END_VAR
VAR_INST
	boolEx				: BoolEx := (variable := _boolVariable);
	conditionTrueTimer	: Tc2_Standard.TON;
END_VAR
TcUnit.TEST('Test01_BooleanTrue_ExpectTrueAfterElapsedTime');

conditionTrueTimer();
IF NOT conditionTrueTimer.Q THEN
	_boolVariable := TRUE;
	conditionTrueTimer(IN := TRUE, PT := T#20MS);
	AssertFalse(
		Condition := boolEx.HasBeenTrueForAtLeast(T#20MS),
		Message := 'HasBeenTrueForAtLeast returned TRUE before elapsed time.');
ELSE
	AssertTrue(
		Condition := boolEx.HasBeenTrueForAtLeast(T#20MS),
		Message := 'HasBeenTrueForAtLeast returned FALSE after elapsed time.');
		TcUnit.TEST_FINISHED();
END_IF
END_METHOD

METHOD Test02_BooleanFalse_ExpectTrueAfterElapsedTime : BOOL
VAR_INST
	boolEx			: BoolEx := (variable := _boolVariable);
	conditionTimer	: Tc2_Standard.TON;
END_VAR
TcUnit.TEST('Test02_BooleanFalse_ExpectTrueAfterElapsedTime');
IF TcUnit.IS_TEST_FINISHED('Test01_BooleanTrue_ExpectTrueAfterElapsedTime') THEN
	_boolVariable := FALSE;
	conditionTimer();
	IF NOT conditionTimer.Q THEN
		conditionTimer(IN := TRUE, PT := T#20MS);
		AssertFalse(
			Condition := boolEx.HasBeenFalseForAtLeast(T#20MS),
			Message := 'HasBeenFalseForAtLeast returned TRUE before elapsed time.');
	ELSE
		AssertTrue(
			Condition := boolEx.HasBeenFalseForAtLeast(T#20MS),
			Message := 'HasBeenFalseForAtLeast returned FALSE after elapsed time.');
			TcUnit.TEST_FINISHED();
	END_IF
END_IF
END_METHOD

METHOD Test03_RisingAndFallingEdge_ExpectPulses
VAR_INPUT
END_VAR

VAR_INST
	boolEx : BoolEx := (variable := _boolVariable);
END_VAR
TcUnit.TEST('Test03_RisingAndFallingEdge_ExpectPulses');


IF TcUnit.IS_TEST_FINISHED('Test02_BooleanFalse_ExpectTrueAfterElapsedTime') THEN
	_boolVariable := FALSE;
	AssertFalse(
		Condition := boolEx.HasRisingEdge,
		Message := 'When value has not changed, the HasRisingEdge should be false');
	AssertFalse(
		Condition := boolEx.HasFallingEdge,
		Message := 'When value has not changed, the HasFallingEdge should be false');
	_boolVariable := TRUE;	
	AssertTrue(
		Condition := boolEx.HasRisingEdge,
		Message := 'When value has changed from FALSE to TRUE, the HasRisingEdge should be TRUE');
	AssertFalse(
		Condition := boolEx.HasFallingEdge,
		Message := 'When value has changed to TRUE, the HasFallingEdge should be false');
	_boolVariable := FALSE;
	AssertTrue(
		Condition := boolEx.HasFallingEdge,
		Message := 'When value has changed from TRUE to FALSE, the HasFallingEdge should be TRUE');
	AssertFalse(
		Condition := boolEx.HasRisingEdge,
		Message := 'When value has not changed, the HasRisingEdge should be false');
	AssertFalse(
		Condition := boolEx.HasFallingEdge,
		Message := 'When value has not changed, the HasRisingEdge should be false');	
	TcUnit.TEST_FINISHED();
	
END_IF
END_METHOD

METHOD Test04_GetAndSetValue
VAR_INPUT
END_VAR
VAR_INST
	boolEx	: BoolEx := (variable := _boolVariable);
END_VAR
TcUnit.TEST('Test04_GetAndSetValue');
IF TcUnit.IS_TEST_FINISHED('Test03_RisingAndFallingEdge_ExpectPulses') THEN
	_boolVariable := FALSE;
	boolEx.Value := TRUE;	
	AssertTrue(
		Condition := _boolVariable,
		Message := 'Setting value to TRUE failed');
		
	boolEx.Value := FALSE;
	AssertFalse(
		Condition := _boolVariable,
		Message := 'Setting value to FALSE failed');
		
	AssertEquals_BOOL(
		Actual := boolEx.Value,
		Expected := _boolVariable,
		Message := 'Value returned incorrect result.');
		
	_boolVariable := TRUE;
	AssertEquals_BOOL(
		Actual := boolEx.Value,
		Expected := _boolVariable,
		Message := 'Value returned incorrect result.');
	
	TcUnit.TEST_FINISHED();
END_IF
END_METHOD

METHOD Test05_Toggle_ExpectValueInverts
VAR_INPUT
END_VAR
TcUnit.TEST('Test05_Toggle_ExpectValueInverts');
IF TcUnit.IS_TEST_FINISHED('Test04_GetAndSetValue') THEN
	_boolEx.Value := FALSE;
	AssertFalse(
		Condition := _boolEx.Value,
		Message := 'Expected value to be false.');
		
	_boolEx.Toggle();
	AssertTrue(
		Condition := _boolEx.Value,
		Message := 'Toggle to TRUE failed');
		
	_boolEx.Toggle();
	AssertFalse(
		Condition := _boolEx.Value,
		Message := 'Toggle to FALSE failed');	
	TcUnit.TEST_FINISHED();
END_IF
END_METHOD

METHOD Test06_PulseWithInterval_100ms_ExpectValueChangeEvery100ms
VAR_INPUT
END_VAR
VAR_INST
	timerOn		: Tc2_Standard.TON;
	timerOff	: Tc2_Standard.TON;
END_VAR
TcUnit.TEST('Test06_PulseWithInterval_100ms_ExpectValueChangeEvery100ms');
IF TcUnit.IS_TEST_FINISHED('Test05_Toggle_ExpectValueInverts') THEN
	_boolEx.Value := FALSE;
	_boolEx.PulseWithInterval(durationOn := T#100MS, durationOff := T#50MS);
	timerOn(IN := TRUE, PT := T#100MS);
	IF NOT timerOn.Q THEN
		AssertTrue(
			Condition := _boolEx.Value,
			Message := 'Value should be TRUE until the durationOn expires.');
	ELSE
		timerOff(IN := TRUE, PT := T#50MS);
		IF timeroff.Q THEN
			AssertTrue(
				Condition := _boolEx.Value,
				Message := 'Value should be TRUE after the durationOff expires.');
			TcUnit.TEST_FINISHED();
			RETURN;
		END_IF
		AssertFalse(
			Condition := _boolEx.Value,
			Message := 'Value should be FALSE after durationOn expires.');

	END_IF
END_IF
END_METHOD

METHOD Test07_Set_ExpectTrue
VAR_INPUT
END_VAR
TcUnit.TEST('Test07_Set_ExpectTrue');

IF TcUnit.IS_TEST_FINISHED('Test06_PulseWithInterval_100ms_ExpectValueChangeEvery100ms') THEN 
	_boolEx.Value := FALSE;
	_boolEx.Set();
	AssertTrue(
		Condition := _boolEx.Value,
		Message := 'Set() did not set the value to TRUE.');
	TcUnit.TEST_FINISHED();
END_IF
END_METHOD

METHOD Test08_Reset_ExpectFalse
VAR_INPUT
END_VAR
TcUnit.TEST('Test08_Reset_ExpectFalse');

IF TcUnit.IS_TEST_FINISHED('Test07_Set_ExpectTrue') THEN 
	_boolEx.Value := TRUE;
	_boolEx.Reset();
	AssertFalse(
		Condition := _boolEx.Value,
		Message := 'Reset() did not set the value to FALSE.');
	TcUnit.TEST_FINISHED();
END_IF
END_METHOD

END_FUNCTION_BLOCK

// TESTS/Test suites/FB_DateTimeToStringConverter_Tests
FUNCTION_BLOCK INTERNAL FB_DateTimeToStringConverter_Tests EXTENDS FB_TestSuite
VAR_INPUT
END_VAR
VAR_OUTPUT
END_VAR
VAR
	_localSystemTime			: Tc2_Utilities.FB_LocalSystemTime;
	_dateTimeToStringConverter	: FB_DateTimeToStringConverter;
END_VAR

_localSystemTime(
	sNetID:= '', 
	bEnable:= TRUE, 
	dwCycle:= 1);
	
_dateTimeToStringConverter(localSystemTime := _localSystemTime);

Test01_Year();
Test02_Month();
Test03_Day();
Test04_Hour();
Test05_Minute();
Test06_Second();
Test07_Millisecond();

METHOD Test01_Year
VAR_INPUT
END_VAR
TcUnit.TEST('Test01_Year');

AssertEquals_STRING(
	Actual := _dateTimeToStringConverter.Year(),
	Expected := WORD_TO_STRING(_localSystemTime.systemTime.wYear),
	Message := 'Conversion to string for year was incorrect!');
	
TcUnit.TEST_FINISHED();
END_METHOD

METHOD Test02_Month
VAR_INPUT
END_VAR

VAR
	expected	: STRING;
END_VAR
TcUnit.TEST('Test02_Month');

expected := WORD_TO_STRING(_localSystemTime.systemTime.wMonth);

AssertEquals_STRING(
	Actual := _dateTimeToStringConverter.Month(fillWithZeros := FALSE),
	Expected := expected,
	Message := 'Conversion to string for month without zeros was incorrect!');
	
IF LEN(expected) = 1 THEN
	expected := CONCAT('0', WORD_TO_STRING(_localSystemTime.systemTime.wMonth));
END_IF

AssertEquals_STRING(
	Expected := expected,
	Actual := _dateTimeToStringConverter.Month(fillWithZeros := TRUE),
	Message := 'Conversion to string for month with zeros was incorrect!');
	
TcUnit.TEST_FINISHED();
END_METHOD

METHOD PUBLIC Test03_Day

VAR
	expected : STRING;
END_VAR
TcUnit.TEST('Test03_Day');

expected := WORD_TO_STRING(_localSystemTime.systemTime.wDay);

AssertEquals_STRING(
	Actual := _dateTimeToStringConverter.Day(fillWithZeros := FALSE),
	Expected := expected,
	Message := 'Conversion to string for day without zeros was incorrect!');
	
IF LEN(expected) = 1 THEN
	expected := CONCAT('0', WORD_TO_STRING(_localSystemTime.systemTime.wDay));
END_IF

AssertEquals_STRING(
	Expected := expected,
	Actual := _dateTimeToStringConverter.Day(fillWithZeros := TRUE),
	Message := 'Conversion to string for day with zeros was incorrect!');
	
TcUnit.TEST_FINISHED();
END_METHOD

METHOD PUBLIC Test04_Hour

VAR
	expected : STRING;
END_VAR
TcUnit.TEST('Test04_Hour');

expected := WORD_TO_STRING(_localSystemTime.systemTime.wHour);

AssertEquals_STRING(
	Actual := _dateTimeToStringConverter.Hour(fillWithZeros := FALSE),
	Expected := expected,
	Message := 'Conversion to string for hour without zeros was incorrect!');
	
IF LEN(expected) = 1 THEN
	expected := CONCAT('0', WORD_TO_STRING(_localSystemTime.systemTime.wHour));
END_IF

AssertEquals_STRING(
	Expected := expected,
	Actual := _dateTimeToStringConverter.Hour(fillWithZeros := TRUE),
	Message := 'Conversion to string for hour with zeros was incorrect!');
	
TcUnit.TEST_FINISHED();
END_METHOD

METHOD PUBLIC Test05_Minute

VAR
	expected : STRING;
END_VAR
TcUnit.TEST('Test05_Minute');

expected := WORD_TO_STRING(_localSystemTime.systemTime.wMinute);

AssertEquals_STRING(
	Actual := _dateTimeToStringConverter.Minute(fillWithZeros := FALSE),
	Expected := expected,
	Message := 'Conversion to string for minute without zeros was incorrect!');
	
IF LEN(expected) = 1 THEN
	expected := CONCAT('0', WORD_TO_STRING(_localSystemTime.systemTime.wMinute));
END_IF

AssertEquals_STRING(
	Expected := expected,
	Actual := _dateTimeToStringConverter.Minute(fillWithZeros := TRUE),
	Message := 'Conversion to string for minute with zeros was incorrect!');
	
TcUnit.TEST_FINISHED();
END_METHOD

METHOD PUBLIC Test06_Second

VAR
	expected : STRING;
END_VAR
TcUnit.TEST('Test06_Second');

expected := WORD_TO_STRING(_localSystemTime.systemTime.wSecond);

AssertEquals_STRING(
	Actual := _dateTimeToStringConverter.Second(fillWithZeros := FALSE),
	Expected := expected,
	Message := 'Conversion to string for second without zeros was incorrect!');
	
IF LEN(expected) = 1 THEN
	expected := CONCAT('0', WORD_TO_STRING(_localSystemTime.systemTime.wSecond));
END_IF

AssertEquals_STRING(
	Expected := expected,
	Actual := _dateTimeToStringConverter.Second(fillWithZeros := TRUE),
	Message := 'Conversion to string for second with zeros was incorrect!');
	
TcUnit.TEST_FINISHED();
END_METHOD

METHOD PUBLIC Test07_Millisecond

VAR
	expected : STRING;
END_VAR
TcUnit.TEST('Test07_Millisecond');

expected := WORD_TO_STRING(_localSystemTime.systemTime.wMilliseconds);

AssertEquals_STRING(
	Actual := _dateTimeToStringConverter.Millisecond(fillWithZeros := FALSE),
	Expected := expected,
	Message := 'Conversion to string for millisecond without zeros was incorrect!');
	
IF LEN(expected) = 1 THEN
	expected := CONCAT('0', WORD_TO_STRING(_localSystemTime.systemTime.wMilliseconds));
END_IF

AssertEquals_STRING(
	Expected := expected,
	Actual := _dateTimeToStringConverter.Second(fillWithZeros := TRUE),
	Message := 'Conversion to string for millisecond with zeros was incorrect!');
	
TcUnit.TEST_FINISHED();
END_METHOD

END_FUNCTION_BLOCK

// TESTS/Test suites/FB_ErrorSource_ExtensionForTests
// Since FB_ErrorSource is an ABSTRACT class, the functionality needs to be implemented by extending the base class
FUNCTION_BLOCK INTERNAL FB_ErrorSource_ExtensionForTests EXTENDS FB_ErrorSource
VAR_INPUT
	eAdsErrorCodeToTest 	: TcError.AdsErrorCodes;
	sGenericErrorMessage	: Tc2_System.T_MaxString;
	nGenericErrorCode		: DINT;
	bError					: BOOL;		
END_VAR

THIS^.AdsError.Code := eAdsErrorCodeToTest;
THIS^.GenericError.Message := sGenericErrorMessage;
THIS^.GenericError.Code := nGenericErrorCode;
THIS^.Error := bError;

END_FUNCTION_BLOCK

// TESTS/Test suites/FB_ErrorSource_Tests
FUNCTION_BLOCK INTERNAL FB_ErrorSource_Tests EXTENDS FB_TestSuite
VAR_INPUT
END_VAR
VAR_OUTPUT
END_VAR
VAR
	_errorSourceObject	: FB_ErrorSource_ExtensionForTests;
END_VAR

Test01_ErrorProperty();
Test02_ErrorCode();
Test03_ErrorMessage();
Test04_GenericError();

METHOD Test01_ErrorProperty
VAR_INPUT
END_VAR
TcUnit.TEST('Test01_ErrorProperty');
_errorSourceObject.bError := TRUE;
_errorSourceObject();
AssertTrue(
	Condition := _errorSourceObject.Error,
	Message := 'Error should be TRUE.');	
	
TcUnit.TEST_FINISHED();
END_METHOD

METHOD Test02_ErrorCode
VAR
END_VAR
TcUnit.TEST('Test02_ErrorCode');

_errorSourceObject.eAdsErrorCodeToTest := TcError.AdsErrorCodes.ADSERR_CLIENT_ERROR;
_errorSourceObject();

AssertEquals_UDINT(
	Actual := _errorSourceObject.AdsError.Code,
	Expected := TcError.AdsErrorCodes.ADSERR_CLIENT_ERROR,
	Message := 'The error code provided in the ErrorInfo.Code property is incorrect!');

TcUnit.TEST_FINISHED();
END_METHOD

METHOD PRIVATE Test03_ErrorMessage
VAR_INPUT
END_VAR
TcUnit.TEST('Test03_ErrorMessage');

_errorSourceObject.eAdsErrorCodeToTest := TcError.AdsErrorCodes.ADSERR_DEVICE_ABORTED;
_errorSourceObject();

AssertEquals_STRING(
	Actual := _errorSourceObject.AdsError.Message,
	Expected := 'Request is aborted.',
	Message := 'The error information was incorrect!');

TcUnit.TEST_FINISHED();
END_METHOD

METHOD Test04_GenericError
VAR_INPUT
END_VAR
TcUnit.TEST('Test04_GenericError');

_errorSourceObject.nGenericErrorCode := 10;
_errorSourceObject.sGenericErrorMessage := 'Error message, generic...';
_errorSourceObject();
AssertEquals_DINT(
	Expected := 10,
	Actual := _errorSourceObject.GenericError.Code,
	Message := 'Incorrect error code.');
	
AssertEquals_STRING(
	Expected := 'Error message, generic...',
	Actual := _errorSourceObject.GenericError.Message,
	Message := 'Incorrect error message.');
	
TcUnit.TEST_FINISHED();
END_METHOD

END_FUNCTION_BLOCK

// TESTS/Test suites/FB_EthercatHelper_Tests
FUNCTION_BLOCK INTERNAL FB_EthercatHelper_Tests EXTENDS FB_TestSuite
VAR_INPUT
END_VAR
VAR_OUTPUT
END_VAR
VAR
END_VAR

Test01_ConvertBeckhoffEcState_ProvideAllOptions_ExpectCorrectResults();

METHOD Test01_ConvertBeckhoffEcState_ProvideAllOptions_ExpectCorrectResults
VAR_INST
	ecSlaveState		: Tc2_EtherCAT.ST_EcSlaveState;
	helperEcSlaveState	: ST_EcSlaveState;
END_VAR
TcUnit.TEST('Test01_ConvertBeckhoffEcState_ProvideAllOptions_ExpectCorrectResults');

// Init
ecSlaveState.deviceState := Tc2_EtherCAT.EC_DEVICE_STATE_INIT;
helperEcSlaveState := EthercatHelper.ConvertBeckhoffEcStateToCustomStruct(ecSlaveState);
AssertEquals_BYTE(Tc2_EtherCAT.EC_DEVICE_STATE_INIT, helperEcSlaveState.Device.State, 'Incorrect state for EC_DEVICE_STATE_INIT.');
AssertEquals_BYTE(E_EcDeviceStateExtras.NOTHING, helperEcSlaveState.Device.StateExtras, 'EC_DEVICE_STATE_INIT - Extras NOTHING expected');
	
ecSlaveState.deviceState := Tc2_EtherCAT.EC_DEVICE_STATE_INIT OR Tc2_EtherCAT.EC_DEVICE_STATE_INITCMD_ERROR;
helperEcSlaveState := EthercatHelper.ConvertBeckhoffEcStateToCustomStruct(ecSlaveState);
AssertEquals_BYTE(Tc2_EtherCAT.EC_DEVICE_STATE_INIT, helperEcSlaveState.Device.State,'Incorrect state for EC_DEVICE_STATE_INIT OR EC_DEVICE_STATE_INITCMD_ERROR');
AssertEquals_BYTE(E_EcDeviceStateExtras.INIIT_CMD_ERROR, helperEcSlaveState.Device.StateExtras, 'EC_DEVICE_STATE_INIT - Extras INIIT_CMD_ERROR expected');
	
ecSlaveState.deviceState := Tc2_EtherCAT.EC_DEVICE_STATE_INIT OR Tc2_EtherCAT.EC_DEVICE_STATE_INVALID_VPRS;
helperEcSlaveState := EthercatHelper.ConvertBeckhoffEcStateToCustomStruct(ecSlaveState);
AssertEquals_BYTE(Tc2_EtherCAT.EC_DEVICE_STATE_INIT, helperEcSlaveState.Device.State,'Incorrect state for EC_DEVICE_STATE_INIT OR EC_DEVICE_STATE_INVALID_VPRS');
AssertEquals_BYTE(E_EcDeviceStateExtras.INVALID_VPRS, helperEcSlaveState.Device.StateExtras, 'EC_DEVICE_STATE_INIT - Extras INVALID_VPRS expected');

ecSlaveState.deviceState := Tc2_EtherCAT.EC_DEVICE_STATE_INIT OR Tc2_EtherCAT.EC_DEVICE_STATE_DISABLED;
helperEcSlaveState := EthercatHelper.ConvertBeckhoffEcStateToCustomStruct(ecSlaveState);
AssertEquals_BYTE(Tc2_EtherCAT.EC_DEVICE_STATE_INIT, helperEcSlaveState.Device.State,'Incorrect state for EC_DEVICE_STATE_INIT OR EC_DEVICE_STATE_DISABLED');
AssertEquals_BYTE(E_EcDeviceStateExtras.DISABLED, helperEcSlaveState.Device.StateExtras, 'EC_DEVICE_STATE_INIT - Extras DISABLED expected');

ecSlaveState.deviceState := Tc2_EtherCAT.EC_DEVICE_STATE_INIT OR Tc2_EtherCAT.EC_DEVICE_STATE_ERROR;
helperEcSlaveState := EthercatHelper.ConvertBeckhoffEcStateToCustomStruct(ecSlaveState);
AssertEquals_BYTE(Tc2_EtherCAT.EC_DEVICE_STATE_INIT, helperEcSlaveState.Device.State,'Incorrect state for EC_DEVICE_STATE_INIT OR EC_DEVICE_STATE_ERROR');
AssertEquals_BYTE(E_EcDeviceStateExtras.STATE_MACHINE_ERROR, helperEcSlaveState.Device.StateExtras, 'EC_DEVICE_STATE_INIT - Extras STATE_MACHINE_ERROR expected');
	
// Pre-op
ecSlaveState.deviceState := Tc2_EtherCAT.EC_DEVICE_STATE_PREOP;
helperEcSlaveState := EthercatHelper.ConvertBeckhoffEcStateToCustomStruct(ecSlaveState);
AssertEquals_BYTE(Tc2_EtherCAT.EC_DEVICE_STATE_PREOP, helperEcSlaveState.Device.State, 'Incorrect state for EC_DEVICE_STATE_PREOP.');
AssertEquals_BYTE(E_EcDeviceStateExtras.NOTHING, helperEcSlaveState.Device.StateExtras, 'EC_DEVICE_STATE_PREOP - Extras NOTHING expected');
	
ecSlaveState.deviceState := Tc2_EtherCAT.EC_DEVICE_STATE_PREOP OR Tc2_EtherCAT.EC_DEVICE_STATE_INITCMD_ERROR;
helperEcSlaveState := EthercatHelper.ConvertBeckhoffEcStateToCustomStruct(ecSlaveState);
AssertEquals_BYTE(Tc2_EtherCAT.EC_DEVICE_STATE_PREOP, helperEcSlaveState.Device.State,'Incorrect state for EC_DEVICE_STATE_PREOP OR EC_DEVICE_STATE_INITCMD_ERROR');
AssertEquals_BYTE(E_EcDeviceStateExtras.INIIT_CMD_ERROR, helperEcSlaveState.Device.StateExtras, 'EC_DEVICE_STATE_PREOP - Extras INIIT_CMD_ERROR expected');
	
ecSlaveState.deviceState := Tc2_EtherCAT.EC_DEVICE_STATE_PREOP OR Tc2_EtherCAT.EC_DEVICE_STATE_INVALID_VPRS;
helperEcSlaveState := EthercatHelper.ConvertBeckhoffEcStateToCustomStruct(ecSlaveState);
AssertEquals_BYTE(Tc2_EtherCAT.EC_DEVICE_STATE_PREOP, helperEcSlaveState.Device.State,'Incorrect state for EC_DEVICE_STATE_PREOP OR EC_DEVICE_STATE_INVALID_VPRS');
AssertEquals_BYTE(E_EcDeviceStateExtras.INVALID_VPRS, helperEcSlaveState.Device.StateExtras, 'EC_DEVICE_STATE_PREOP - Extras INVALID_VPRS expected');

ecSlaveState.deviceState := Tc2_EtherCAT.EC_DEVICE_STATE_PREOP OR Tc2_EtherCAT.EC_DEVICE_STATE_DISABLED;
helperEcSlaveState := EthercatHelper.ConvertBeckhoffEcStateToCustomStruct(ecSlaveState);
AssertEquals_BYTE(Tc2_EtherCAT.EC_DEVICE_STATE_PREOP, helperEcSlaveState.Device.State,'Incorrect state for EC_DEVICE_STATE_PREOP OR EC_DEVICE_STATE_DISABLED');
AssertEquals_BYTE(E_EcDeviceStateExtras.DISABLED, helperEcSlaveState.Device.StateExtras, 'EC_DEVICE_STATE_PREOP - Extras DISABLED expected');

ecSlaveState.deviceState := Tc2_EtherCAT.EC_DEVICE_STATE_PREOP OR Tc2_EtherCAT.EC_DEVICE_STATE_ERROR;
helperEcSlaveState := EthercatHelper.ConvertBeckhoffEcStateToCustomStruct(ecSlaveState);
AssertEquals_BYTE(Tc2_EtherCAT.EC_DEVICE_STATE_PREOP, helperEcSlaveState.Device.State,'Incorrect state for EC_DEVICE_STATE_PREOP OR EC_DEVICE_STATE_ERROR');
AssertEquals_BYTE(E_EcDeviceStateExtras.STATE_MACHINE_ERROR, helperEcSlaveState.Device.StateExtras, 'EC_DEVICE_STATE_PREOP - Extras STATE_MACHINE_ERROR expected');

// Bootstrap
ecSlaveState.deviceState := Tc2_EtherCAT.EC_DEVICE_STATE_BOOTSTRAP;
helperEcSlaveState := EthercatHelper.ConvertBeckhoffEcStateToCustomStruct(ecSlaveState);
AssertEquals_BYTE(Tc2_EtherCAT.EC_DEVICE_STATE_BOOTSTRAP, helperEcSlaveState.Device.State, 'Incorrect state for EC_DEVICE_STATE_BOOTSTRAP.');
AssertEquals_BYTE(E_EcDeviceStateExtras.NOTHING, helperEcSlaveState.Device.StateExtras, 'EC_DEVICE_STATE_BOOTSTRAP - Extras NOTHING expected');
	
ecSlaveState.deviceState := Tc2_EtherCAT.EC_DEVICE_STATE_BOOTSTRAP OR Tc2_EtherCAT.EC_DEVICE_STATE_INITCMD_ERROR;
helperEcSlaveState := EthercatHelper.ConvertBeckhoffEcStateToCustomStruct(ecSlaveState);
AssertEquals_BYTE(Tc2_EtherCAT.EC_DEVICE_STATE_BOOTSTRAP, helperEcSlaveState.Device.State,'Incorrect state for EC_DEVICE_STATE_BOOTSTRAP OR EC_DEVICE_STATE_INITCMD_ERROR');
AssertEquals_BYTE(E_EcDeviceStateExtras.INIIT_CMD_ERROR, helperEcSlaveState.Device.StateExtras, 'EC_DEVICE_STATE_BOOTSTRAP - Extras INIIT_CMD_ERROR expected');
	
ecSlaveState.deviceState := Tc2_EtherCAT.EC_DEVICE_STATE_BOOTSTRAP OR Tc2_EtherCAT.EC_DEVICE_STATE_INVALID_VPRS;
helperEcSlaveState := EthercatHelper.ConvertBeckhoffEcStateToCustomStruct(ecSlaveState);
AssertEquals_BYTE(Tc2_EtherCAT.EC_DEVICE_STATE_BOOTSTRAP, helperEcSlaveState.Device.State,'Incorrect state for EC_DEVICE_STATE_BOOTSTRAP OR EC_DEVICE_STATE_INVALID_VPRS');
AssertEquals_BYTE(E_EcDeviceStateExtras.INVALID_VPRS, helperEcSlaveState.Device.StateExtras, 'EC_DEVICE_STATE_BOOTSTRAP - Extras INVALID_VPRS expected');

ecSlaveState.deviceState := Tc2_EtherCAT.EC_DEVICE_STATE_BOOTSTRAP OR Tc2_EtherCAT.EC_DEVICE_STATE_DISABLED;
helperEcSlaveState := EthercatHelper.ConvertBeckhoffEcStateToCustomStruct(ecSlaveState);
AssertEquals_BYTE(Tc2_EtherCAT.EC_DEVICE_STATE_BOOTSTRAP, helperEcSlaveState.Device.State,'Incorrect state for EC_DEVICE_STATE_BOOTSTRAP OR EC_DEVICE_STATE_DISABLED');
AssertEquals_BYTE(E_EcDeviceStateExtras.DISABLED, helperEcSlaveState.Device.StateExtras, 'EC_DEVICE_STATE_BOOTSTRAP - Extras DISABLED expected');

ecSlaveState.deviceState := Tc2_EtherCAT.EC_DEVICE_STATE_BOOTSTRAP OR Tc2_EtherCAT.EC_DEVICE_STATE_ERROR;
helperEcSlaveState := EthercatHelper.ConvertBeckhoffEcStateToCustomStruct(ecSlaveState);
AssertEquals_BYTE(Tc2_EtherCAT.EC_DEVICE_STATE_BOOTSTRAP, helperEcSlaveState.Device.State,'Incorrect state for EC_DEVICE_STATE_BOOTSTRAP OR EC_DEVICE_STATE_ERROR');
AssertEquals_BYTE(E_EcDeviceStateExtras.STATE_MACHINE_ERROR, helperEcSlaveState.Device.StateExtras, 'EC_DEVICE_STATE_BOOTSTRAP - Extras STATE_MACHINE_ERROR expected');

// Safeop
ecSlaveState.deviceState := Tc2_EtherCAT.EC_DEVICE_STATE_SAFEOP;
helperEcSlaveState := EthercatHelper.ConvertBeckhoffEcStateToCustomStruct(ecSlaveState);
AssertEquals_BYTE(Tc2_EtherCAT.EC_DEVICE_STATE_SAFEOP, helperEcSlaveState.Device.State, 'Incorrect state for EC_DEVICE_STATE_SAFEOP.');
AssertEquals_BYTE(E_EcDeviceStateExtras.NOTHING, helperEcSlaveState.Device.StateExtras, 'EC_DEVICE_STATE_SAFEOP - Extras NOTHING expected');
	
ecSlaveState.deviceState := Tc2_EtherCAT.EC_DEVICE_STATE_SAFEOP OR Tc2_EtherCAT.EC_DEVICE_STATE_INITCMD_ERROR;
helperEcSlaveState := EthercatHelper.ConvertBeckhoffEcStateToCustomStruct(ecSlaveState);
AssertEquals_BYTE(Tc2_EtherCAT.EC_DEVICE_STATE_SAFEOP, helperEcSlaveState.Device.State,'Incorrect state for EC_DEVICE_STATE_BOOTSTRAP OR EC_DEVICE_STATE_INITCMD_ERROR');
AssertEquals_BYTE(E_EcDeviceStateExtras.INIIT_CMD_ERROR, helperEcSlaveState.Device.StateExtras, 'EC_DEVICE_STATE_SAFEOP - Extras INIIT_CMD_ERROR expected');
	
ecSlaveState.deviceState := Tc2_EtherCAT.EC_DEVICE_STATE_SAFEOP OR Tc2_EtherCAT.EC_DEVICE_STATE_INVALID_VPRS;
helperEcSlaveState := EthercatHelper.ConvertBeckhoffEcStateToCustomStruct(ecSlaveState);
AssertEquals_BYTE(Tc2_EtherCAT.EC_DEVICE_STATE_SAFEOP, helperEcSlaveState.Device.State,'Incorrect state for EC_DEVICE_STATE_SAFEOP OR EC_DEVICE_STATE_INVALID_VPRS');
AssertEquals_BYTE(E_EcDeviceStateExtras.INVALID_VPRS, helperEcSlaveState.Device.StateExtras, 'EC_DEVICE_STATE_SAFEOP - Extras INVALID_VPRS expected');

ecSlaveState.deviceState := Tc2_EtherCAT.EC_DEVICE_STATE_SAFEOP OR Tc2_EtherCAT.EC_DEVICE_STATE_DISABLED;
helperEcSlaveState := EthercatHelper.ConvertBeckhoffEcStateToCustomStruct(ecSlaveState);
AssertEquals_BYTE(Tc2_EtherCAT.EC_DEVICE_STATE_SAFEOP, helperEcSlaveState.Device.State,'Incorrect state for EC_DEVICE_STATE_SAFEOP OR EC_DEVICE_STATE_DISABLED');
AssertEquals_BYTE(E_EcDeviceStateExtras.DISABLED, helperEcSlaveState.Device.StateExtras, 'EC_DEVICE_STATE_SAFEOP - Extras DISABLED expected');

ecSlaveState.deviceState := Tc2_EtherCAT.EC_DEVICE_STATE_SAFEOP OR Tc2_EtherCAT.EC_DEVICE_STATE_ERROR;
helperEcSlaveState := EthercatHelper.ConvertBeckhoffEcStateToCustomStruct(ecSlaveState);
AssertEquals_BYTE(Tc2_EtherCAT.EC_DEVICE_STATE_SAFEOP, helperEcSlaveState.Device.State,'Incorrect state for EC_DEVICE_STATE_SAFEOP OR EC_DEVICE_STATE_ERROR');
AssertEquals_BYTE(E_EcDeviceStateExtras.STATE_MACHINE_ERROR, helperEcSlaveState.Device.StateExtras, 'EC_DEVICE_STATE_SAFEOP - Extras STATE_MACHINE_ERROR expected');

// OP
ecSlaveState.deviceState := Tc2_EtherCAT.EC_DEVICE_STATE_OP;
helperEcSlaveState := EthercatHelper.ConvertBeckhoffEcStateToCustomStruct(ecSlaveState);
AssertEquals_BYTE(Tc2_EtherCAT.EC_DEVICE_STATE_OP, helperEcSlaveState.Device.State, 'Incorrect state for EC_DEVICE_STATE_OP.');
AssertEquals_BYTE(E_EcDeviceStateExtras.NOTHING, helperEcSlaveState.Device.StateExtras, 'EC_DEVICE_STATE_OP - Extras NOTHING expected');
	
ecSlaveState.deviceState := Tc2_EtherCAT.EC_DEVICE_STATE_OP OR Tc2_EtherCAT.EC_DEVICE_STATE_INITCMD_ERROR;
helperEcSlaveState := EthercatHelper.ConvertBeckhoffEcStateToCustomStruct(ecSlaveState);
AssertEquals_BYTE(Tc2_EtherCAT.EC_DEVICE_STATE_OP, helperEcSlaveState.Device.State,'Incorrect state for EC_DEVICE_STATE_OP OR EC_DEVICE_STATE_INITCMD_ERROR');
AssertEquals_BYTE(E_EcDeviceStateExtras.INIIT_CMD_ERROR, helperEcSlaveState.Device.StateExtras, 'EC_DEVICE_STATE_OP - Extras INIIT_CMD_ERROR expected');
	
ecSlaveState.deviceState := Tc2_EtherCAT.EC_DEVICE_STATE_OP OR Tc2_EtherCAT.EC_DEVICE_STATE_INVALID_VPRS;
helperEcSlaveState := EthercatHelper.ConvertBeckhoffEcStateToCustomStruct(ecSlaveState);
AssertEquals_BYTE(Tc2_EtherCAT.EC_DEVICE_STATE_OP, helperEcSlaveState.Device.State,'Incorrect state for EC_DEVICE_STATE_OP OR EC_DEVICE_STATE_INVALID_VPRS');
AssertEquals_BYTE(E_EcDeviceStateExtras.INVALID_VPRS, helperEcSlaveState.Device.StateExtras, 'EC_DEVICE_STATE_OP - Extras INVALID_VPRS expected');

ecSlaveState.deviceState := Tc2_EtherCAT.EC_DEVICE_STATE_OP OR Tc2_EtherCAT.EC_DEVICE_STATE_DISABLED;
helperEcSlaveState := EthercatHelper.ConvertBeckhoffEcStateToCustomStruct(ecSlaveState);
AssertEquals_BYTE(Tc2_EtherCAT.EC_DEVICE_STATE_OP, helperEcSlaveState.Device.State,'Incorrect state for EC_DEVICE_STATE_OP OR EC_DEVICE_STATE_DISABLED');
AssertEquals_BYTE(E_EcDeviceStateExtras.DISABLED, helperEcSlaveState.Device.StateExtras, 'EC_DEVICE_STATE_OP - Extras DISABLED expected');

ecSlaveState.deviceState := Tc2_EtherCAT.EC_DEVICE_STATE_OP OR Tc2_EtherCAT.EC_DEVICE_STATE_ERROR;
helperEcSlaveState := EthercatHelper.ConvertBeckhoffEcStateToCustomStruct(ecSlaveState);
AssertEquals_BYTE(Tc2_EtherCAT.EC_DEVICE_STATE_OP, helperEcSlaveState.Device.State,'Incorrect state for EC_DEVICE_STATE_OP OR EC_DEVICE_STATE_ERROR');
AssertEquals_BYTE(E_EcDeviceStateExtras.STATE_MACHINE_ERROR, helperEcSlaveState.Device.StateExtras, 'EC_DEVICE_STATE_OP - Extras STATE_MACHINE_ERROR expected');

// Link state

//EC_LINK_STATE_OK
ecSlaveState.linkState := Tc2_EtherCAT.EC_LINK_STATE_OK;
helperEcSlaveState := EthercatHelper.ConvertBeckhoffEcStateToCustomStruct(ecSlaveState);
AssertEquals_BYTE(Tc2_EtherCAT.EC_LINK_STATE_OK, helperEcSlaveState.Link, 'Invalid link state for EC_LINK_STATE_OK');

// EC_LINK_STATE_ADDITIONAL_LINK
ecSlaveState.linkState := Tc2_EtherCAT.EC_LINK_STATE_ADDITIONAL_LINK;
helperEcSlaveState := EthercatHelper.ConvertBeckhoffEcStateToCustomStruct(ecSlaveState);
AssertEquals_BYTE(E_EcLinkState.ADDITIONAL_LINK, helperEcSlaveState.Link, 'Invalid link state for EC_LINK_STATE_ADDITIONAL_LINK');

// EC_LINK_STATE_LINK_WITHOUT_COMM
ecSlaveState.linkState := Tc2_EtherCAT.EC_LINK_STATE_LINK_WITHOUT_COMM;
helperEcSlaveState := EthercatHelper.ConvertBeckhoffEcStateToCustomStruct(ecSlaveState);
AssertEquals_BYTE(E_EcLinkState.LINK_WITHOUT_COMM, helperEcSlaveState.Link, 'Invalid link state for EC_LINK_STATE_LINK_WITHOUT_COMM');

// EC_LINK_STATE_MISSING_LINK
ecSlaveState.linkState := Tc2_EtherCAT.EC_LINK_STATE_MISSING_LINK;
helperEcSlaveState := EthercatHelper.ConvertBeckhoffEcStateToCustomStruct(ecSlaveState);
AssertEquals_BYTE(E_EcLinkState.MISSING_LINK, helperEcSlaveState.Link, 'Invalid link state for EC_LINK_STATE_MISSING_LINK');

// EC_LINK_STATE_NOT_PRESENT
ecSlaveState.linkState := Tc2_EtherCAT.EC_LINK_STATE_NOT_PRESENT;
helperEcSlaveState := EthercatHelper.ConvertBeckhoffEcStateToCustomStruct(ecSlaveState);
AssertEquals_BYTE(E_EcLinkState.NOT_PRESENT, helperEcSlaveState.Link, 'Invalid link state for EC_LINK_STATE_NOT_PRESENT');

// EC_LINK_STATE_PORT_A
ecSlaveState.linkState := Tc2_EtherCAT.EC_LINK_STATE_PORT_A;
helperEcSlaveState := EthercatHelper.ConvertBeckhoffEcStateToCustomStruct(ecSlaveState);
AssertEquals_BYTE(E_EcLinkState.PORT_A, helperEcSlaveState.Link, 'Invalid link state for EC_LINK_STATE_PORT_A');

// EC_LINK_STATE_PORT_B
ecSlaveState.linkState := Tc2_EtherCAT.EC_LINK_STATE_PORT_B;
helperEcSlaveState := EthercatHelper.ConvertBeckhoffEcStateToCustomStruct(ecSlaveState);
AssertEquals_BYTE(E_EcLinkState.PORT_B, helperEcSlaveState.Link, 'Invalid link state for EC_LINK_STATE_PORT_B');

// EC_LINK_STATE_PORT_C
ecSlaveState.linkState := Tc2_EtherCAT.EC_LINK_STATE_PORT_C;
helperEcSlaveState := EthercatHelper.ConvertBeckhoffEcStateToCustomStruct(ecSlaveState);
AssertEquals_BYTE(E_EcLinkState.PORT_C, helperEcSlaveState.Link, 'Invalid link state for EC_LINK_STATE_PORT_C');

// EC_LINK_STATE_PORT_D
ecSlaveState.linkState := Tc2_EtherCAT.EC_LINK_STATE_PORT_D;
helperEcSlaveState := EthercatHelper.ConvertBeckhoffEcStateToCustomStruct(ecSlaveState);
AssertEquals_BYTE(E_EcLinkState.PORT_D, helperEcSlaveState.Link, 'Invalid link state for EC_LINK_STATE_PORT_D');

TcUnit.TEST_FINISHED();
END_METHOD

END_FUNCTION_BLOCK

// TESTS/Test suites/FB_HasInstanceName_ExtensionForTests
// Since FB_HasInstanceName is an ABSTRACT class, 
// the functionality needs to be implemented by extending the base class
FUNCTION_BLOCK INTERNAL FB_HasInstanceName_ExtensionForTests EXTENDS FB_HasInstanceNameAndPath
VAR_INPUT
END_VAR
VAR_OUTPUT
END_VAR
VAR
END_VAR

END_FUNCTION_BLOCK

// TESTS/Test suites/FB_HasInstanceName_Tests
FUNCTION_BLOCK INTERNAL FB_HasInstanceName_Tests EXTENDS FB_TestSuite
VAR_INPUT
END_VAR
VAR_OUTPUT
END_VAR
VAR
	fbHasInstanceName	:  FB_HasInstanceName_ExtensionForTests;
END_VAR

Test01_InstanceName();
Test02_InstancePath();

METHOD Test01_InstanceName
VAR_INPUT
END_VAR
TcUnit.TEST('Test01_InstanceName');

AssertEquals_STRING(
	Expected := 'fbHasInstanceName',
	Actual := fbHasInstanceName.InstanceName,
	Message := 'InstanceName is not correct.');
	
TcUnit.TEST_FINISHED();
END_METHOD

METHOD Test02_InstancePath
VAR_INPUT
END_VAR
TcUnit.TEST('Test02_InstancePath');

AssertEquals_STRING(
	Expected := 'PRG_TESTS.HasInstanceNameTests.fbHasInstanceName',
	Actual := fbHasInstanceName.InstancePath,
	Message := 'Instance path is incorrect.');

TcUnit.TEST_FINISHED();
END_METHOD

END_FUNCTION_BLOCK

// TESTS/PRG_TESTS
PROGRAM INTERNAL PRG_TESTS

(* Instantiate test suites here. Naming convention for tests should be a suffix with _Tests.
Good practice for creating test methods is to end them with _test as well. *)
VAR
	AdsHelperTests					: FB_AdsHelper_Tests;
	ArrayHelperTests				: FB_ArrayHelper_Tests;
	DateTimeToStringConverterTest	: FB_DateTimeToStringConverter_Tests;
	ErrorSourceTests				: FB_ErrorSource_Tests;
	HasInstanceNameTests			: FB_HasInstanceName_Tests;
	StringBuilderTests				: FB_StringBuilder_Tests;
	HasTaskInfoTests				: FB_HasTaskInfo_Tests;
	BoolExTests						: FB_BoolEx_Tests;
	EthercatHelperTests				: FB_EthercatHelper_Tests;
	//EthercatDiagnosisTests			: FB_EthercatDiagnosis_Tests;
	MallocTests						: FB_Malloc_Tests;
	StringHelperTests				: FB_StringHelper_Tests;
	LocalSystemTimeTests			: FB_LocalSystemTime_Tests;
END_VAR

// Run tests in paralel
//TcUnit.RUN();

// Run tests in sequence, one after the other. Uncomment if required.
TcUnit.RUN_IN_SEQUENCE();

END_PROGRAM

// TESTS/Test suites/FB_StringBuilder_Tests
FUNCTION_BLOCK INTERNAL FB_StringBuilder_Tests EXTENDS FB_StringBuilderEx_Any_Tests
VAR_INPUT
END_VAR
VAR_OUTPUT
END_VAR
VAR
	_stringBuilder	: FB_StringBuilder;
END_VAR

Test01_AddStrings_ExpectConcat();
Test02_AddWithSingleQuotationMarks();
Test03_AddWithDoubleQuotationMarks();
Test04_CreateDoesNotResetStringSequence();
Test05_ResetClearsBuildSequence();
SUPER^();

METHOD Test01_AddStrings_ExpectConcat
VAR_INPUT
END_VAR
IF TcUnit.TEST_ORDERED('Test01_AddStrings_ExpectConcat') THEN
	AssertEquals_STRING(
		Actual := _stringBuilder.Reset()
			.AddString('test')
			.AddString('test2')
			.Create(),
		Expected := 'testtest2',
		Message := 'AddString of two strings failed!');
		
	TcUnit.TEST_FINISHED();
END_IF
END_METHOD

METHOD Test02_AddWithSingleQuotationMarks
VAR_INPUT
END_VAR
IF TcUnit.TEST_ORDERED('Test02_AddWithSingleQuotationMarks') THEN
	AssertEquals_STRING(
		Actual := _stringBuilder.Reset()
			.AddWithQuotationMark('test')
			.AddWithQuotationMark('test2')
			.Create(),
		Expected := '$'test$'$'test2$'',
		Message := 'AddString of two strings failed!');
		
	TcUnit.TEST_FINISHED();
END_IF
END_METHOD

METHOD Test03_AddWithDoubleQuotationMarks
VAR_INPUT
END_VAR
IF TcUnit.TEST_ORDERED('Test03_AddWithDoubleQuotationMarks') THEN
	AssertEquals_STRING(
		Actual := _stringBuilder.Reset()
			.AddWithDblQuotationMarks('test')
			.AddWithDblQuotationMarks('test2')
			.Create(),
		Expected := '"test""test2"',
		Message := 'AddString of two strings failed!');
		
	TcUnit.TEST_FINISHED();
END_IF
END_METHOD

METHOD Test04_CreateDoesNotResetStringSequence
VAR_INPUT
END_VAR
IF TcUnit.TEST_ORDERED('Test04_CreateDoesNotResetStringSequence') THEN
	_stringBuilder.Reset()
		.AddString('a')
		.AddString('b')
		.Create();
		
	AssertEquals_STRING(
		Actual := _stringBuilder.AddString('c').Create(),
		Expected := 'abc',
		Message := 'Calling .Create() should result in the string creation remaining intact, until Reset() is called explicitly!');
		
	TcUnit.TEST_FINISHED();
END_IF
END_METHOD

METHOD Test05_ResetClearsBuildSequence
VAR_INPUT
END_VAR
IF TcUnit.TEST_ORDERED('Test05_ResetClearsBuildSequence') THEN
	_stringBuilder.Reset()
		.AddString('a')
		.AddString('b')
		.Reset()
		.AddString('c');
	
	AssertEquals_STRING(
		Actual := _stringBuilder.Create(),
		Expected := 'c',
		Message := 'Calling Reset() method should result in the sequnce being cleared!');
		
	TcUnit.TEST_FINISHED();
END_IF
END_METHOD

END_FUNCTION_BLOCK

// TESTS/Test suites/FB_StringBuilderEx_Any_Tests
FUNCTION_BLOCK INTERNAL FB_StringBuilderEx_Any_Tests EXTENDS TcUnit.FB_TestSuite
VAR_INPUT
END_VAR
VAR_OUTPUT
END_VAR
VAR
	stringBuilder	: FB_StringBuilder;
END_VAR

Test01_BOOL();
Test02_BYTE();
Test03_DATE();
Test04_DateAndTime();
Test05_DINT();
Test06_DWORD();
Test07_ENUM();
Test08_INT();
Test09_LINT();
Test10_LREAL();
Test11_LTIME();
Test12_LWORD();
Test13_REAL();
Test14_SINT();
Test15_STRING();
Test16_TIME();
Test17_TOD();
Test18_UDINT();
Test19_UINT();
Test20_ULINT();
Test21_USINT();
Test22_WORD();
Test23_WSTRING();
Test24_ANY_BIT_WORD();
Test25_ANY_BIT_BYTE();
Test26_ANY_BIT_DWORD();
Test27_ANY_BIT_LWORD();
Test28_ANY_REAL_REAL();
Test29_ANY_REAL_LREAL();

METHOD Test01_BOOL
VAR_INPUT
END_VAR

VAR_INST
	bTrue		: BOOL := TRUE;
	bFalse		: BOOL := FALSE;

END_VAR
IF TcUnit.TEST_ORDERED('Test01_BOOL') THEN
	AssertEquals_STRING(
		Actual := stringBuilder.Reset().AddAny(bTrue).Create(),
		Expected := 'TRUE',
		Message := 'Adding boolean failed');
		
	AssertEquals_STRING(
		Actual := stringBuilder.Reset().AddAny(bFalse).Create(),
		Expected := 'FALSE',
		Message := 'Adding boolean failed');
		
	TcUnit.TEST_FINISHED();
END_IF
END_METHOD

METHOD Test02_BYTE
VAR_INPUT
END_VAR
VAR
	byteVar	: BYTE := 17;
END_VAR
IF TEST_ORDERED('Test02_BYTE') THEN
	
	AssertEquals_STRING(
		Actual := stringBuilder.Reset().AddAny(byteVar).Create(),
		Expected := '17',
		Message := 'Adding BYTE failed.');
	TEST_FINISHED();
END_IF
END_METHOD

METHOD Test03_DATE
VAR
	someVar	: DATE := D#1970-01-01;
END_VAR
IF TEST_ORDERED('Test03_DATE') THEN
	AssertEquals_STRING(
		Actual := stringBuilder.Reset().AddAny(someVar).Create(),
		Expected := 'D#1970-01-01',
		Message := 'Adding DATE failed.');

	TEST_FINISHED();
END_IF
END_METHOD

METHOD Test04_DateAndTime
VAR
	someVar	: DATE_AND_TIME := DT#1970-1-1-0:0:1;
END_VAR
IF TEST_ORDERED('Test04_DateAndTime') THEN
	AssertEquals_STRING(
		Actual := stringBuilder.Reset().AddAny(someVar).Create(),
		Expected := 'DT#1970-01-01-00:00:01',
		Message := 'Adding DATE_AND_TIME failed.');

	TEST_FINISHED();
END_IF
END_METHOD

METHOD Test05_DINT
VAR
	someVar	: DINT := 15;
END_VAR
IF TEST_ORDERED('Test05_DINT') THEN
	AssertEquals_STRING(
		Actual := stringBuilder.Reset().AddAny(someVar).Create(),
		Expected := '15',
		Message := 'Adding DINT failed.');

	TEST_FINISHED();
END_IF
END_METHOD

METHOD Test06_DWORD
VAR
	someVar	: DWORD := 777;
END_VAR
IF TEST_ORDERED('Test06_DWORD') THEN
	AssertEquals_STRING(
		Actual := stringBuilder.Reset().AddAny(someVar).Create(),
		Expected := '777',
		Message := 'Adding DWORD failed.');

	TEST_FINISHED();
END_IF
END_METHOD

METHOD Test07_ENUM
VAR
	someVar	: E_AddAnyBitOptions := E_AddAnyBitOptions.HEXADECIMAL;
END_VAR
IF TEST_ORDERED('Test07_ENUM') THEN
	AssertEquals_STRING(
		Actual := stringBuilder.Reset().AddAny(someVar).Create(),
		Expected := '2',
		Message := 'Adding ENUM failed.');

	TEST_FINISHED();
END_IF
END_METHOD

METHOD Test08_INT
VAR
	someVar	: INT := 22;
END_VAR
IF TEST_ORDERED('Test08_INT') THEN
	AssertEquals_STRING(
		Actual := stringBuilder.Reset().AddAny(someVar).Create(),
		Expected := '22',
		Message := 'Adding INT failed.');

	TEST_FINISHED();
END_IF
END_METHOD

METHOD Test09_LINT
VAR
	someVar	: LINT := 6666;
END_VAR
IF TEST_ORDERED('Test09_LINT') THEN
	AssertEquals_STRING(
		Actual := stringBuilder.Reset().AddAny(someVar).Create(),
		Expected := '6666',
		Message := 'Adding LINT failed.');

	TEST_FINISHED();
END_IF
END_METHOD

METHOD Test10_LREAL
VAR
	someVar	: LREAL := 11.11;
END_VAR
IF TEST_ORDERED('Test10_LREAL') THEN
	AssertEquals_STRING(
		Actual := stringBuilder.Reset().AddAny(someVar).Create(),
		Expected := '11.11',
		Message := 'Adding LREAL failed.');

	TEST_FINISHED();
END_IF
END_METHOD

METHOD Test11_LTIME
VAR
	someVar	: LTIME := LTIME#100D2H30M40S500MS600US700NS;
END_VAR
IF TEST_ORDERED('Test11_LTIME') THEN
	AssertEquals_STRING(
		Actual := stringBuilder.Reset().AddAny(someVar).Create(),
		Expected := 'LTIME#100d2h30m40s500ms600us700ns',
		Message := 'Adding LTIME failed.');

	TEST_FINISHED();
END_IF
END_METHOD

METHOD Test12_LWORD
VAR
	someVar	: LWORD := 123456;
END_VAR
IF TEST_ORDERED('Test12_LWORD') THEN
	AssertEquals_STRING(
		Actual := stringBuilder.Reset().AddAny(someVar).Create(),
		Expected := '123456',
		Message := 'Adding LWORD failed.');

	TEST_FINISHED();
END_IF
END_METHOD

METHOD Test13_REAL
VAR
	someVar	: REAL := 12345.6789;
END_VAR
IF TEST_ORDERED('Test13_REAL') THEN
	AssertEquals_STRING(
		Actual := stringBuilder.Reset().AddAny(someVar).Create(),
		Expected := '12345.679',
		Message := 'Adding REAL failed.');

	TEST_FINISHED();
END_IF
END_METHOD

METHOD Test14_SINT
VAR
	someVar	: SINT := -34;
END_VAR
IF TEST_ORDERED('Test14_SINT') THEN
	AssertEquals_STRING(
		Actual := stringBuilder.Reset().AddAny(someVar).Create(),
		Expected := '-34',
		Message := 'Adding SINT failed.');

	TEST_FINISHED();
END_IF
END_METHOD

METHOD Test15_STRING
VAR
	someVar	: STRING := 'haha';
END_VAR
IF TEST_ORDERED('Test15_STRING') THEN
	AssertEquals_STRING(
		Actual := stringBuilder.Reset().AddAny(someVar).Create(),
		Expected := 'haha',
		Message := 'Adding STRING failed.');

	TEST_FINISHED();
END_IF
END_METHOD

METHOD Test16_TIME
VAR
	someVar	: TIME := T#15D10S;
END_VAR
IF TEST_ORDERED('Test16_TIME') THEN
	AssertEquals_STRING(
		Actual := stringBuilder.Reset().AddAny(someVar).Create(),
		Expected := 'T#15d10s',
		Message := 'Adding TIME failed.');

	TEST_FINISHED();
END_IF
END_METHOD

METHOD Test17_TOD
VAR
	someVar	: TOD := TOD#14:01:05.123;
END_VAR
IF TEST_ORDERED('Test17_TOD') THEN
	AssertEquals_STRING(
		Actual := stringBuilder.Reset().AddAny(someVar).Create(),
		Expected := 'TOD#14:01:05.123',
		Message := 'Adding TOD failed.');

	TEST_FINISHED();
END_IF
END_METHOD

METHOD Test18_UDINT
VAR
	someVar	: UDINT := 23452352;
END_VAR
IF TEST_ORDERED('Test18_UDINT') THEN
	AssertEquals_STRING(
		Actual := stringBuilder.Reset().AddAny(someVar).Create(),
		Expected := '23452352',
		Message := 'Adding UDINT failed.');

	TEST_FINISHED();
END_IF
END_METHOD

METHOD Test19_UINT
VAR
	someVar	: UINT := 12341;
END_VAR
IF TEST_ORDERED('Test19_UINT') THEN
	AssertEquals_STRING(
		Actual := stringBuilder.Reset().AddAny(someVar).Create(),
		Expected := '12341',
		Message := 'Adding UINT failed.');

	TEST_FINISHED();
END_IF
END_METHOD

METHOD Test20_ULINT
VAR
	someVar	: ULINT := 12345678;
END_VAR
IF TEST_ORDERED('Test20_ULINT') THEN
	AssertEquals_STRING(
		Actual := stringBuilder.Reset().AddAny(someVar).Create(),
		Expected := '12345678',
		Message := 'Adding ULINT failed.');

	TEST_FINISHED();
END_IF
END_METHOD

METHOD Test21_USINT
VAR
	someVar	: USINT := 123;
END_VAR
IF TEST_ORDERED('Test21_USINT') THEN
	AssertEquals_STRING(
		Actual := stringBuilder.Reset().AddAny(someVar).Create(),
		Expected := '123',
		Message := 'Adding USINT failed.');

	TEST_FINISHED();
END_IF
END_METHOD

METHOD Test22_WORD
VAR
	someVar	: WORD := 16#A;
END_VAR
IF TEST_ORDERED('Test22_WORD') THEN
	AssertEquals_STRING(
		Actual := stringBuilder.Reset().AddAny(someVar).Create(),
		Expected := '10',
		Message := 'Adding WORD failed.');

	TEST_FINISHED();
END_IF
END_METHOD

METHOD Test23_WSTRING
VAR
	someVar	: WSTRING := "test";
END_VAR
IF TEST_ORDERED('Test23_WSTRING') THEN
	AssertEquals_STRING(
		Actual := stringBuilder.Reset().AddAny(someVar).Create(),
		Expected := 'test',
		Message := 'Adding WSTRING failed.');

	TEST_FINISHED();
END_IF
END_METHOD

METHOD Test24_ANY_BIT_WORD
VAR_INPUT
END_VAR
VAR
	wordVar	: WORD := 16#AB;
	result	: Tc2_System.T_MaxString;
END_VAR
IF TcUnit.TEST_ORDERED('Test24_ANY_BIT_WORD') THEN
	
	// BINARY with notations
	result := stringBuilder.Reset().
		AddAnyBit(
			anyBit := wordVar, 
			option := E_AddAnyBitOptions.BINARY, 
			lowerCase := FALSE, 
			displayedDigitsCount := 16, 
			addNotation := TRUE)
		.Create();
		
	AssertEquals_STRING(
		Actual := result,
		Expected := '(BIN)0000000010101011',
		Message := 'Adding word as BINARY with addNotation = TRUE was incorrect');
		
	// BINARY without notations
	result := stringBuilder.Reset()
		.AddAnyBit(
			anyBit := wordVar, 
			option := E_AddAnyBitOptions.BINARY, 
			lowerCase := FALSE, 
			displayedDigitsCount := 16, 
			addNotation := FALSE)
		.Create();
		
	AssertEquals_STRING(
		Actual := result,
		Expected := '0000000010101011',
		Message := 'Adding word as BINARY with addNotation = FALSE was incorrect');
		
	// DECIMAL with notations
	result := stringBuilder.Reset()
		.AddAnyBit(
			anyBit := wordVar, 
			option := E_AddAnyBitOptions.DECIMAL, 
			lowerCase := FALSE, 
			displayedDigitsCount := 16, 
			addNotation := TRUE)
		.Create();
		
	AssertEquals_STRING(
		Actual := result,
		Expected := '(DEC)0000000000000171',
		Message := 'Adding word as DECIMAL with addNotation = TRUE was incorrect');
		
	// DECIMAL without notations
	result := stringBuilder.Reset()
		.AddAnyBit(
			anyBit := wordVar, 
			option := E_AddAnyBitOptions.DECIMAL, 
			lowerCase := FALSE, 
			displayedDigitsCount := 16, 
			addNotation := FALSE)
		.Create();
		
	AssertEquals_STRING(
		Actual := result,
		Expected := '0000000000000171',
		Message := 'Adding word as DECIMAL with addNotation = FALSE was incorrect');

	// HEXADECIMAL with notations
	result := stringBuilder.Reset()
		.AddAnyBit(
			anyBit := wordVar, 
			option := E_AddAnyBitOptions.HEXADECIMAL, 
			lowerCase := FALSE, 
			displayedDigitsCount := 16, 
			addNotation := TRUE)
		.Create();
		
	AssertEquals_STRING(
		Actual := result,
		Expected := '(HEX)00000000000000AB',
		Message := 'Adding word as HEXADECIMAL with addNotation = TRUE was incorrect');
		
	// HEXADECIMAL without notations
	result := stringBuilder.Reset()
		.AddAnyBit(
			anyBit := wordVar, 
			option := E_AddAnyBitOptions.HEXADECIMAL, 
			lowerCase := FALSE, 
			displayedDigitsCount := 16, 
			addNotation := FALSE)
		.Create();
		
	AssertEquals_STRING(
		Actual := result,
		Expected := '00000000000000AB',
		Message := 'Adding word as HEXADECIMAL with addNotation = FALSE was incorrect');
	
	// OCTAL with notations
	result := stringBuilder.Reset()
		.AddAnyBit(
			anyBit := wordVar, 
			option := E_AddAnyBitOptions.OCTAL, 
			lowerCase := FALSE, 
			displayedDigitsCount := 16, 
			addNotation := TRUE)
		.Create();
		
	AssertEquals_STRING(
		Actual := result,
		Expected := '(OCT)0000000000000253',
		Message := 'Adding word as OCTAL with addNotation = TRUE was incorrect');
		
	// OCTAL without notations
	result := stringBuilder.Reset()
		.AddAnyBit(
			anyBit := wordVar, 
			option := E_AddAnyBitOptions.OCTAL, 
			lowerCase := FALSE, 
			displayedDigitsCount := 16, 
			addNotation := FALSE)
		.Create();
		
	AssertEquals_STRING(
		Actual := result,
		Expected := '0000000000000253',
		Message := 'Adding word as OCTAL with addNotation = FALSE was incorrect');
		
	TcUnit.TEST_FINISHED();
END_IF
END_METHOD

METHOD Test25_ANY_BIT_BYTE
VAR_INPUT
END_VAR
VAR
	byteVar	: BYTE := 16#AB;
	result	: Tc2_System.T_MaxString;
END_VAR
IF TcUnit.TEST_ORDERED('Test25_ANY_BIT_BYTE') THEN
	
	// BINARY with notations
	result := stringBuilder.Reset().
		AddAnyBit(
			anyBit := byteVar, 
			option := E_AddAnyBitOptions.BINARY, 
			lowerCase := FALSE, 
			displayedDigitsCount := 8, 
			addNotation := TRUE)
		.Create();
		
	AssertEquals_STRING(
		Actual := result,
		Expected := '(BIN)10101011',
		Message := 'Adding byte as BINARY with addNotation = TRUE was incorrect');
		
	// BINARY without notations
	result := stringBuilder.Reset()
		.AddAnyBit(
			anyBit := byteVar, 
			option := E_AddAnyBitOptions.BINARY, 
			lowerCase := FALSE, 
			displayedDigitsCount := 8, 
			addNotation := FALSE)
		.Create();
		
	AssertEquals_STRING(
		Actual := result,
		Expected := '10101011',
		Message := 'Adding byte as BINARY with addNotation = FALSE was incorrect');
		
	// DECIMAL with notations
	result := stringBuilder.Reset()
		.AddAnyBit(
			anyBit := byteVar, 
			option := E_AddAnyBitOptions.DECIMAL, 
			lowerCase := FALSE, 
			displayedDigitsCount := 8, 
			addNotation := TRUE)
		.Create();
		
	AssertEquals_STRING(
		Actual := result,
		Expected := '(DEC)00000171',
		Message := 'Adding byte as DECIMAL with addNotation = TRUE was incorrect');
		
	// DECIMAL without notations
	result := stringBuilder.Reset()
		.AddAnyBit(
			anyBit := byteVar, 
			option := E_AddAnyBitOptions.DECIMAL, 
			lowerCase := FALSE, 
			displayedDigitsCount := 8, 
			addNotation := FALSE)
		.Create();
		
	AssertEquals_STRING(
		Actual := result,
		Expected := '00000171',
		Message := 'Adding byte as DECIMAL with addNotation = FALSE was incorrect');

	// HEXADECIMAL with notations
	result := stringBuilder.Reset()
		.AddAnyBit(
			anyBit := byteVar, 
			option := E_AddAnyBitOptions.HEXADECIMAL, 
			lowerCase := FALSE, 
			displayedDigitsCount := 8, 
			addNotation := TRUE)
		.Create();
		
	AssertEquals_STRING(
		Actual := result,
		Expected := '(HEX)000000AB',
		Message := 'Adding byte as HEXADECIMAL with addNotation = TRUE was incorrect');
		
	// HEXADECIMAL without notations
	result := stringBuilder.Reset()
		.AddAnyBit(
			anyBit := byteVar, 
			option := E_AddAnyBitOptions.HEXADECIMAL, 
			lowerCase := FALSE, 
			displayedDigitsCount := 8, 
			addNotation := FALSE)
		.Create();
		
	AssertEquals_STRING(
		Actual := result,
		Expected := '000000AB',
		Message := 'Adding byte as HEXADECIMAL with addNotation = FALSE was incorrect');
	
	// OCTAL with notations
	result := stringBuilder.Reset()
		.AddAnyBit(
			anyBit := byteVar, 
			option := E_AddAnyBitOptions.OCTAL, 
			lowerCase := FALSE, 
			displayedDigitsCount := 8, 
			addNotation := TRUE)
		.Create();
		
	AssertEquals_STRING(
		Actual := result,
		Expected := '(OCT)00000253',
		Message := 'Adding byte as OCTAL with addNotation = TRUE was incorrect');
		
	// OCTAL without notations
	result := stringBuilder.Reset()
		.AddAnyBit(
			anyBit := byteVar, 
			option := E_AddAnyBitOptions.OCTAL, 
			lowerCase := FALSE, 
			displayedDigitsCount := 8, 
			addNotation := FALSE)
		.Create();
		
	AssertEquals_STRING(
		Actual := result,
		Expected := '00000253',
		Message := 'Adding byte as OCTAL with addNotation = FALSE was incorrect');
		
	TcUnit.TEST_FINISHED();
END_IF
END_METHOD

METHOD Test26_ANY_BIT_DWORD
VAR
	dwordVar	: DWORD := 16#AB;
	result	: Tc2_System.T_MaxString;
END_VAR
IF TcUnit.TEST_ORDERED('Test26_ANY_BIT_DWORD') THEN
	
	// BINARY with notations
	result := stringBuilder.Reset().
		AddAnyBit(
			anyBit := dwordVar, 
			option := E_AddAnyBitOptions.BINARY, 
			lowerCase := FALSE, 
			displayedDigitsCount := 32, 
			addNotation := TRUE)
		.Create();
		
	AssertEquals_STRING(
		Actual := result,
		Expected := '(BIN)00000000000000000000000010101011',
		Message := 'Adding dword as BINARY with addNotation = TRUE was incorrect');
		
	// BINARY without notations
	result := stringBuilder.Reset()
		.AddAnyBit(
			anyBit := dwordVar, 
			option := E_AddAnyBitOptions.BINARY, 
			lowerCase := FALSE, 
			displayedDigitsCount := 32, 
			addNotation := FALSE)
		.Create();
		
	AssertEquals_STRING(
		Actual := result,
		Expected := '00000000000000000000000010101011',
		Message := 'Adding dword as BINARY with addNotation = FALSE was incorrect');
		
	// DECIMAL with notations
	result := stringBuilder.Reset()
		.AddAnyBit(
			anyBit := dwordVar, 
			option := E_AddAnyBitOptions.DECIMAL, 
			lowerCase := FALSE, 
			displayedDigitsCount := 32, 
			addNotation := TRUE)
		.Create();
		
	AssertEquals_STRING(
		Actual := result,
		Expected := '(DEC)00000000000000000000000000000171',
		Message := 'Adding dword as DECIMAL with addNotation = TRUE was incorrect');
		
	// DECIMAL without notations
	result := stringBuilder.Reset()
		.AddAnyBit(
			anyBit := dwordVar, 
			option := E_AddAnyBitOptions.DECIMAL, 
			lowerCase := FALSE, 
			displayedDigitsCount := 32, 
			addNotation := FALSE)
		.Create();
		
	AssertEquals_STRING(
		Actual := result,
		Expected := '00000000000000000000000000000171',
		Message := 'Adding dword as DECIMAL with addNotation = FALSE was incorrect');

	// HEXADECIMAL with notations
	result := stringBuilder.Reset()
		.AddAnyBit(
			anyBit := dwordVar, 
			option := E_AddAnyBitOptions.HEXADECIMAL, 
			lowerCase := FALSE, 
			displayedDigitsCount := 32, 
			addNotation := TRUE)
		.Create();
		
	AssertEquals_STRING(
		Actual := result,
		Expected := '(HEX)000000000000000000000000000000AB',
		Message := 'Adding dword as HEXADECIMAL with addNotation = TRUE was incorrect');
		
	// HEXADECIMAL without notations
	result := stringBuilder.Reset()
		.AddAnyBit(
			anyBit := dwordVar, 
			option := E_AddAnyBitOptions.HEXADECIMAL, 
			lowerCase := FALSE, 
			displayedDigitsCount := 32, 
			addNotation := FALSE)
		.Create();
		
	AssertEquals_STRING(
		Actual := result,
		Expected := '000000000000000000000000000000AB',
		Message := 'Adding dword as HEXADECIMAL with addNotation = FALSE was incorrect');
	
	// OCTAL with notations
	result := stringBuilder.Reset()
		.AddAnyBit(
			anyBit := dwordVar, 
			option := E_AddAnyBitOptions.OCTAL, 
			lowerCase := FALSE, 
			displayedDigitsCount := 32, 
			addNotation := TRUE)
		.Create();
		
	AssertEquals_STRING(
		Actual := result,
		Expected := '(OCT)00000000000000000000000000000253',
		Message := 'Adding dword as OCTAL with addNotation = TRUE was incorrect');
		
	// OCTAL without notations
	result := stringBuilder.Reset()
		.AddAnyBit(
			anyBit := dwordVar, 
			option := E_AddAnyBitOptions.OCTAL, 
			lowerCase := FALSE, 
			displayedDigitsCount := 32, 
			addNotation := FALSE)
		.Create();
		
	AssertEquals_STRING(
		Actual := result,
		Expected := '00000000000000000000000000000253',
		Message := 'Adding dword as OCTAL with addNotation = FALSE was incorrect');
		
	TcUnit.TEST_FINISHED();
END_IF
END_METHOD

METHOD Test27_ANY_BIT_LWORD
VAR
	lwordVar	: LWORD := 16#AB;
	result	: Tc2_System.T_MaxString;
END_VAR
IF TcUnit.TEST_ORDERED('Test27_ANY_BIT_LWORD') THEN
	
	// BINARY with notations
	result := stringBuilder.Reset().
		AddAnyBit(
			anyBit := lwordVar, 
			option := E_AddAnyBitOptions.BINARY, 
			lowerCase := FALSE, 
			displayedDigitsCount := 64, 
			addNotation := TRUE)
		.Create();
		
	AssertEquals_STRING(
		Actual := result,
		Expected := '(BIN)0000000000000000000000000000000000000000000000000000000010101011',
		Message := 'Adding lword as BINARY with addNotation = TRUE was incorrect');
		
	// BINARY without notations
	result := stringBuilder.Reset()
		.AddAnyBit(
			anyBit := lwordVar, 
			option := E_AddAnyBitOptions.BINARY, 
			lowerCase := FALSE, 
			displayedDigitsCount := 64, 
			addNotation := FALSE)
		.Create();
		
	AssertEquals_STRING(
		Actual := result,
		Expected := '0000000000000000000000000000000000000000000000000000000010101011',
		Message := 'Adding lword as BINARY with addNotation = FALSE was incorrect');
		
	// DECIMAL with notations
	result := stringBuilder.Reset()
		.AddAnyBit(
			anyBit := lwordVar, 
			option := E_AddAnyBitOptions.DECIMAL, 
			lowerCase := FALSE, 
			displayedDigitsCount := 64, 
			addNotation := TRUE)
		.Create();
		
	AssertEquals_STRING(
		Actual := result,
		Expected := '(DEC)0000000000000000000000000000000000000000000000000000000000000171',
		Message := 'Adding lword as DECIMAL with addNotation = TRUE was incorrect');
		
	// DECIMAL without notations
	result := stringBuilder.Reset()
		.AddAnyBit(
			anyBit := lwordVar, 
			option := E_AddAnyBitOptions.DECIMAL, 
			lowerCase := FALSE, 
			displayedDigitsCount := 64, 
			addNotation := FALSE)
		.Create();
		
	AssertEquals_STRING(
		Actual := result,
		Expected := '0000000000000000000000000000000000000000000000000000000000000171',
		Message := 'Adding lword as DECIMAL with addNotation = FALSE was incorrect');

	// HEXADECIMAL with notations
	result := stringBuilder.Reset()
		.AddAnyBit(
			anyBit := lwordVar, 
			option := E_AddAnyBitOptions.HEXADECIMAL, 
			lowerCase := FALSE, 
			displayedDigitsCount := 64, 
			addNotation := TRUE)
		.Create();
		
	AssertEquals_STRING(
		Actual := result,
		Expected := '(HEX)00000000000000000000000000000000000000000000000000000000000000AB',
		Message := 'Adding lword as HEXADECIMAL with addNotation = TRUE was incorrect');
		
	// HEXADECIMAL without notations
	result := stringBuilder.Reset()
		.AddAnyBit(
			anyBit := lwordVar, 
			option := E_AddAnyBitOptions.HEXADECIMAL, 
			lowerCase := FALSE, 
			displayedDigitsCount := 64, 
			addNotation := FALSE)
		.Create();
		
	AssertEquals_STRING(
		Actual := result,
		Expected := '00000000000000000000000000000000000000000000000000000000000000AB',
		Message := 'Adding lword as HEXADECIMAL with addNotation = FALSE was incorrect');
	
	// OCTAL with notations
	result := stringBuilder.Reset()
		.AddAnyBit(
			anyBit := lwordVar, 
			option := E_AddAnyBitOptions.OCTAL, 
			lowerCase := FALSE, 
			displayedDigitsCount := 64, 
			addNotation := TRUE)
		.Create();
		
	AssertEquals_STRING(
		Actual := result,
		Expected := '(OCT)0000000000000000000000000000000000000000000000000000000000000253',
		Message := 'Adding lword as OCTAL with addNotation = TRUE was incorrect');
		
	// OCTAL without notations
	result := stringBuilder.Reset()
		.AddAnyBit(
			anyBit := lwordVar, 
			option := E_AddAnyBitOptions.OCTAL, 
			lowerCase := FALSE, 
			displayedDigitsCount := 64, 
			addNotation := FALSE)
		.Create();
		
	AssertEquals_STRING(
		Actual := result,
		Expected := '0000000000000000000000000000000000000000000000000000000000000253',
		Message := 'Adding lword as OCTAL with addNotation = FALSE was incorrect');
		
	TcUnit.TEST_FINISHED();
END_IF
END_METHOD

METHOD Test28_ANY_REAL_REAL
VAR
	realVar	: REAL := 12345.123888;
	result	: Tc2_System.T_MaxString;
END_VAR
IF TcUnit.TEST_ORDERED('Test28_ANY_REAL_REAL') THEN
	result := stringBuilder.Reset().
		AddAnyReal(
			anyReal := realVar,
			precision := 2,
			round := FALSE)
		.Create();	

	AssertEquals_STRING(
		Actual := result,
		Expected := '12345.12',
		Message := 'Adding REAL with round = FALSE failed.');
		
	result := stringBuilder.Reset().
		AddAnyReal(
			anyReal := realVar,
			precision := 3,
			round := TRUE)
		.Create();	

	AssertEquals_STRING(
		Actual := result,
		Expected := '12345.124',
		Message := 'Adding REAL with round = TRUE failed.');
		
	TcUnit.TEST_FINISHED();
END_IF
END_METHOD

METHOD Test29_ANY_REAL_LREAL
VAR
	lrealVar	: LREAL := 12345.12345678;
	result	: Tc2_System.T_MaxString;
END_VAR
IF TcUnit.TEST_ORDERED('Test29_ANY_REAL_LREAL') THEN
	result := stringBuilder.Reset().
		AddAnyReal(
			anyReal := lrealVar,
			precision := 5,
			round := FALSE)
		.Create();	

	AssertEquals_STRING(
		Actual := result,
		Expected := '12345.12345',
		Message := 'Adding LREAL with round = FALSE failed.');
		
	result := stringBuilder.Reset().
		AddAnyReal(
			anyReal := lrealVar,
			precision := 7,
			round := TRUE)
		.Create();	

	AssertEquals_STRING(
		Actual := result,
		Expected := '12345.1234568',
		Message := 'Adding LREAL with round = TRUE failed.');
		
	TcUnit.TEST_FINISHED();
END_IF
END_METHOD

END_FUNCTION_BLOCK

// TESTS/Test suites/FB_HasTaskInfo_Tests
FUNCTION_BLOCK internal FB_HasTaskInfo_Tests EXTENDS FB_TestSuite
VAR_INPUT
END_VAR
VAR_OUTPUT
END_VAR
VAR
END_VAR

Test01_TaskInfoPropertyValidity();

METHOD Test01_TaskInfoPropertyValidity
VAR_INPUT
END_VAR
VAR_INST
	fbTaskInfo	: FB_HasTaskInfo_ExtensionsForTests;
	cycles	: UINT;
END_VAR
TcUnit.TEST('Test01_TaskInfoPropertyValidity');

AssertTrue(
	Condition := __ISVALIDREF(fbTaskInfo.TaskInfo),
	Message := 'Invalid reference for Taskinfo property. PLC crash will occur if called!');
	
AssertTrue(
	Condition := fbTaskInfo.TaskInfo.AdsPort <> 0,
	Message := 'TaskInfo property is empty.');


TcUnit.TEST_FINISHED();
END_METHOD

END_FUNCTION_BLOCK

// TESTS/Test suites/FB_HasTaskInfo_ExtensionsForTests
// Since FB_HasTaskInfo is an ABSTRACT class, the functionality needs to be implemented by extending the base class
FUNCTION_BLOCK internal FB_HasTaskInfo_ExtensionsForTests EXTENDS FB_HasTaskInfo
VAR_INPUT
END_VAR
VAR_OUTPUT
END_VAR
VAR
END_VAR

END_FUNCTION_BLOCK

// TESTS/Test suites/FB_Malloc_Tests
FUNCTION_BLOCK internal FB_Malloc_Tests EXTENDS FB_TestSuite
VAR_INPUT
END_VAR
VAR_OUTPUT
END_VAR
VAR
	_malloc							: FB_Malloc(0,0);
	_routerInfoBeforeTestMethod		: Tc2_Utilities.ST_TcRouterStatusInfo;
END_VAR

Test01_ProvideIncorrectParameters_ExpectNoAllocation();
Test02_Allocate10Integers_ExpectNoError_ValidateProperties();
Test03_Free_ExpectNoMemoryAllocated();
Test04_SetAndGet_ExpectGetReturnsCorrectValue();
Test05_SetAtIncorrectIndex_ExpectFalseReturned();
Test06_GetFromIncorrectIndex_ExpectTargetValueUnchanged_MethodReturnFalse();
Test07_Expand_ExpectOldDataStillExists_LastDataSetIsEmpty();
Test08_Remove_ExpectDataSetToCollapseBy1();

METHOD BeforeTestFinish : BOOL
VAR_INST
	currentRouterStatus	: Tc2_Utilities.ST_TcRouterStatusInfo;
END_VAR
_malloc.Free();
IF MemoryHelper.GetRouterStatusInfo('', currentRouterStatus) THEN
	AssertEquals_DWORD(
		Expected := _routerInfoBeforeTestMethod.maxMemAvail,
		Actual := currentRouterStatus.maxMemAvail,
		Message := 'The current and starting memory in router differ - memory leak detected.');
	BeforeTestFinish := TRUE;
END_IF
END_METHOD

METHOD BeforeTestStart : BOOL
VAR_INPUT
	methodName	: Tc2_System.T_MaxString;
END_VAR
VAR_INST
	previousMethodName	: Tc2_System.T_MaxString;
	returnValue			: BOOL;
END_VAR
IF previousMethodName <> methodName THEN
	returnValue := FALSE;
END_IF

IF NOT returnValue AND_THEN MemoryHelper.GetRouterStatusInfo('', _routerInfoBeforeTestMethod) THEN
	returnValue := TRUE;
END_IF

previousMethodName := methodName;
BeforeTestStart := returnValue;
END_METHOD

METHOD ValidatePropertiesAfterFailedAllocation
VAR_INPUT
	mallocMethodCalled	: Tc2_System.T_MaxString;
END_VAR
// Validate properties
AssertEquals_DINT(0, _malloc.Properties.BaseTypeSize,
	CONCAT(CONCAT('Calling method ', mallocMethodCalled), ' - BaseTypeSize should be 0 when failing allocation.'));
AssertEquals_DINT(0, _malloc.Properties.NumberOfElements,
	CONCAT(CONCAT('Calling method ', mallocMethodCalled), ' - NumberOfElements should be 0 when failing allocation.'));	
AssertEquals_DINT(0, _malloc.Properties.Size,
	CONCAT(CONCAT('Calling method ', mallocMethodCalled), ' - Size should be 0 when failing allocation.'));			
AssertEquals_ULINT(0, _malloc.Properties.StartAddress,
	CONCAT(CONCAT('Calling method ', mallocMethodCalled), ' - StartAddress should be 0 when failing allocation.'));
END_METHOD

METHOD Test01_ProvideIncorrectParameters_ExpectNoAllocation
VAR_INPUT
END_VAR
VAR
	testMallocVar	: INT;
END_VAR
VAR_INST
	assertionsDone	: BOOL;
END_VAR
IF TcUnit.TEST_ORDERED('Test01_ProvideIncorrectParameters_ExpectNoAllocation') AND_THEN 
	BeforeTestStart('Test01_ProvideIncorrectParameters_ExpectNoAllocation') 
THEN
	IF NOT assertionsDone THEN
		// Manual allocation, element size = 0
		AssertFalse(_malloc.Allocate(0, 10), 
			'If provided size of the element is 0, Allocate should return FALSE.');	
		AssertFalse(_malloc.IsAllocated,
			'IsAllocated property should be false when failing AllocateManual');
		ValidatePropertiesAfterFailedAllocation('Allocate - element size = 0');
		
		// Manual allocation, element count = 0
		AssertFalse(_malloc.Allocate(10, 0),
			'If provided number of elements is 0, Allocat should return FALSE.');	
		AssertFalse(_malloc.IsAllocated,
			'IsAllocated property should be false when failing AllocateManual');
		ValidatePropertiesAfterFailedAllocation('Allocate - element count = 0');
		
		// Manual allocation, element size = -10
		AssertFalse(_malloc.Allocate(-10, 10), 
			'If provided size of the element is -10, AllocateManual should return FALSE.');	
		AssertFalse(_malloc.IsAllocated,
			'IsAllocated property should be false when failing AllocateManual');
		ValidatePropertiesAfterFailedAllocation('Allocate - element size = -10');
		
		// Manual allocation, element count = -10
		AssertFalse(_malloc.Allocate(10, -10),
			'If provided number of elements is -10, Allocate should return FALSE.');	
		AssertFalse(_malloc.IsAllocated,
			'IsAllocated property should be false when failing AllocateManual');
		ValidatePropertiesAfterFailedAllocation('Allocate - element size = -10');
				
		// Any allocation, element count = 0
		AssertFalse(_malloc.AllocateAny(testMallocVar, 0),
			'If provided number of elements is 0, AllocateAny should return FALSE.');	
		AssertFalse(_malloc.IsAllocated,
			'IsAllocated property should be false when failing AllocateManual');		
		ValidatePropertiesAfterFailedAllocation('AllocateAny - element count = 0');
		
		
		// Any allocation, element count = -10
		AssertFalse(_malloc.AllocateAny(testMallocVar, -10),
			'If provided number of elements is 0, AllocateAny should return FALSE.');	
		AssertFalse(_malloc.IsAllocated,
			'IsAllocated property should be false when failing AllocateManual');		
		ValidatePropertiesAfterFailedAllocation('AllocateAny - element count = -10');
		assertionsDone := TRUE;
	END_IF
		
	IF BeforeTestFinish() THEN
		TcUnit.TEST_FINISHED();
	END_IF
END_IF
END_METHOD

METHOD Test02_Allocate10Integers_ExpectNoError_ValidateProperties
VAR_INPUT
END_VAR
VAR_INST
	assertionsDone	: BOOL;
END_VAR
IF TcUnit.TEST_ORDERED('Test02_Allocate10Integers_ExpectNoError_ValidateProperties') AND_THEN 
	BeforeTestStart('Test02_Allocate10Integers_ExpectNoError_ValidateProperties') 
THEN
	IF NOT assertionsDone THEN
		AssertTrue(_malloc.Allocate(SIZEOF(INT), 10),
			'Allocation of 10 integers should return TRUE.');
			
		AssertEquals_DINT(10, _malloc.Properties.NumberOfElements,
			'NumberOfElements is incorrect.');
		AssertEquals_DINT(2, _malloc.Properties.BaseTypeSize,
			'BaseTypeSize  is incorrect.');
		AssertEquals_DINT(10 * 2, _malloc.Properties.Size,
			'Size is incorrect.');
		AssertTrue(_malloc.Properties.StartAddress <> 0,
			'StartAddress should not be 0.');
		assertionsDone := TRUE;
	END_IF
		
	IF BeforeTestFinish() THEN
		TcUnit.TEST_FINISHED();
	END_IF
END_IF
END_METHOD

METHOD Test03_Free_ExpectNoMemoryAllocated
VAR_INPUT
END_VAR
VAR_INST
	assertionsDone	: BOOL;
END_VAR
IF TcUnit.TEST_ORDERED('Test03_Free_ExpectNoMemoryAllocated') AND_THEN 
	BeforeTestStart('Test03_Free_ExpectNoMemoryAllocated') 
THEN
	IF NOT assertionsDone THEN
		_malloc.Allocate(10,10);
		AssertTrue(_malloc.Free(),
			'Freeing allocated memory should return TRUE.');
			
		AssertEquals_DINT(0, _malloc.Properties.NumberOfElements,
			'NumberOfElements should be 0 after freeing.');
		AssertEquals_DINT(0, _malloc.Properties.BaseTypeSize,
			'BaseTypeSize  should be 0 after freeing.');
		AssertEquals_DINT(0, _malloc.Properties.Size,
			'Size should be 0 after freeing.');
		AssertEquals_ULINT(0, _malloc.Properties.StartAddress,
			'StartAddress should be 0 after freeing.');
		AssertFalse(_malloc.IsAllocated,
			'IsAllocated should be FALSE when freeing.');
			
		AssertFalse(_malloc.Free(),
			'If no memory is allocated, Free() should return FALSE.');
		assertionsDone := TRUE;
	END_IF
		
	IF BeforeTestFinish() THEN
		TcUnit.TEST_FINISHED();
	END_IF
END_IF
END_METHOD

METHOD Test04_SetAndGet_ExpectGetReturnsCorrectValue
VAR_INPUT
END_VAR
VAR
	data	: INT;
	result	: INT;
END_VAR
VAR_INST
	assertionsDone	: BOOL;
END_VAR
IF TcUnit.TEST_ORDERED('Test04_SetAndGet_ExpectGetReturnsCorrectValue') AND_THEN 
	BeforeTestStart('Test04_SetAndGet_ExpectGetReturnsCorrectValue') 
THEN
	IF NOT assertionsDone THEN
		_malloc.Allocate(SIZEOF(data), 5);
		
		data := 13;
		AssertTrue(_malloc.Set(2, data), 'Setting value failed.');
			
		_malloc.Get(2, result);
		AssertEquals(data, result, 'Value fetched with Get is not correct.');
		assertionsDone := TRUE;
	END_IF
	
	IF BeforeTestFinish() THEN
		TcUnit.TEST_FINISHED();
	END_IF
END_IF
END_METHOD

METHOD Test05_SetAtIncorrectIndex_ExpectFalseReturned
VAR_INPUT
END_VAR
VAR
	value	: int;
END_VAR
VAR_INST
	assertionsDone	: BOOL;
END_VAR
IF TcUnit.TEST_ORDERED('Test05_SetAtIncorrectIndex_ExpectFalseReturned') AND_THEN 
	BeforeTestStart('Test05_SetAtIncorrectIndex_ExpectFalseReturned') 
THEN
	IF NOT assertionsDone THEN
		_malloc.Allocate(SIZEOF(value),5);
		AssertFalse(_malloc.Set(5, value), 'Setting at index outside range should return FALSE.');	
		assertionsDone := TRUE;
	END_IF
	IF BeforeTestFinish() THEN 
		TcUnit.TEST_FINISHED(); 
	END_IF
END_IF
END_METHOD

METHOD Test06_GetFromIncorrectIndex_ExpectTargetValueUnchanged_MethodReturnFalse
VAR_INPUT
END_VAR

VAR
	result	: INT;
END_VAR
VAR_INST
	assertionsDone	: BOOL;
END_VAR
IF TcUnit.TEST_ORDERED('Test06_GetFromIncorrectIndex_ExpectTargetValueUnchanged_MethodReturnFalse') AND_THEN 
	BeforeTestStart('Test06_GetFromIncorrectIndex_ExpectTargetValueUnchanged_MethodReturnFalse') 
THEN
	IF NOT assertionsDone THEN
		_malloc.AllocateAny(result, 5);
		result := 5;
		AssertFalse(_malloc.Get(5, result), 
			'When getting from index outsied of allocated memory, FALSE should be returned.');
		AssertEquals_int(5,result,
			'Getting from outside the bounds of allocated memory area, result variable should not be changed.');
		assertionsDone := TRUE;
	END_IF
	IF BeforeTestFinish() THEN
		TcUnit.TEST_FINISHED();
	END_IF
END_IF
END_METHOD

METHOD Test07_Expand_ExpectOldDataStillExists_LastDataSetIsEmpty
VAR_INPUT
END_VAR
VAR
	valueToSet	: INT;
	readValue	: INT;
	index		: INT;
END_VAR
VAR_INST
	assertionsDone	: BOOL;
END_VAR
IF TcUnit.TEST_ORDERED('Test07_Expand_ExpectOldDataStillExists_LastDataSetIsEmpty') AND_THEN 
	BeforeTestStart('Test07_Expand_ExpectOldDataStillExists_LastDataSetIsEmpty') 
THEN
	IF NOT assertionsDone THEN
		
		_malloc.Allocate(SIZEOF(INT), 5);
		
		FOR valueToSet := 0 TO 4 BY 1 DO
			_malloc.Set(valueToSet, valueToSet);
			_malloc.get(valueToSet, readValue);
			AssertEquals(
				Actual := readValue,
				Expected := valueToSet,
				Message := 'Incorrect allocation, further tests will fail!');
		END_FOR
		
		_malloc.Expand(3);
		AssertEquals_DINT(
			Actual := _malloc.Properties.NumberOfElements,
			Expected := 8,
			Message := 'Incorrect number of elements after expanding the allocated memory.');
		FOR index := 0 TO 4 BY 1 DO
			_malloc.Get(0,readValue);
			AssertEquals_INT(
				Actual := readValue,
				Expected := readValue,
				Message := Tc2_Standard.CONCAT(TO_STRING(index),'-th element is incorrect after expanding.'));
		END_FOR
		
		_malloc.Get(5, readValue);
		AssertEquals_INT(
			Actual := readValue,
			Expected := 0,
			Message := '5th (new) element is incorrect after expanding.');
			
		_malloc.Get(6, readValue);
		AssertEquals_INT(
			Actual := readValue,
			Expected := 0,
			Message := '6th (new) element is incorrect after expanding.');
			
		_malloc.Get(7, readValue);
		AssertEquals_INT(
			Actual := readValue,
			Expected := 0,
			Message := '7th (new) element is incorrect after expanding.');
		assertionsDone := TRUE;
	END_IF
		
	IF BeforeTestFinish() THEN
		TcUnit.TEST_FINISHED();
	END_IF
END_IF
END_METHOD

METHOD Test08_Remove_ExpectDataSetToCollapseBy1
VAR
	index		: INT;
	readValue	: INT;
END_VAR

VAR_INST
	assertionsDone	: BOOL;
END_VAR
IF TcUnit.TEST_ORDERED('Test08_Remove_ExpectDataSetToCollapseBy1') AND_THEN 
	BeforeTestStart('Test08_Remove_ExpectDataSetToCollapseBy1') 
THEN
	IF NOT assertionsDone THEN
		//[0,1,2,3,4,5]
		_malloc.Allocate(SIZEOF(INT), 6);
		FOR index := 0 TO 5 BY 1 DO
			_malloc.Set(index, index);
			_malloc.Get(index, readValue);
			AssertEquals(Expected := index, Actual := readValue, 
				Message := Tc2_Standard.CONCAT(TO_STRING(index), 'Allocation failed, further tests will fail.'));
		END_FOR
		
		// Expecting //[0,1,2,4,5]
		_malloc.Remove(3);
		AssertEquals_DINT(Expected := 5, Actual := _malloc.Properties.NumberOfElements,
			Message := 'Incorrect number of elements after rmoving the element at index 3.');
	
		_malloc.Get(0, readValue);
		AssertEquals_DINT(Expected := 0, Actual := readValue, 
			Message := '0th element has incorrect value after deleting element at 3rd index.');	
		
		_malloc.Get(1, readValue);
		AssertEquals_DINT(Expected := 1, Actual := readValue, 
			Message := '1st element has incorrect value after deleting element at 3rd index.');	
		
		_malloc.Get(2, readValue);
		AssertEquals_DINT(Expected := 2, Actual := readValue, 
			Message := '2d element has incorrect value after deleting element AT 3rd index.');	
			
			
		_malloc.Get(3, readValue);
		AssertEquals_DINT(Expected := 4, Actual := readValue, 
			Message := '3d element has incorrect value after deleting element AT 3rd index - did allocation not collapse correctly?');	
		
		_malloc.Get(4, readValue);
		AssertEquals_DINT(Expected := 5, Actual := readValue, 
			Message := '4th element has incorrect value after deleting element AT 3rd index - did allocation not collapse correctly?');	
		assertionsDone := TRUE;
	END_IF
	
	IF BeforeTestFinish() THEN
		TcUnit.TEST_FINISHED();
	END_IF
END_IF
END_METHOD

END_FUNCTION_BLOCK

// TESTS/Test suites/FB_StringHelper_Tests
FUNCTION_BLOCK INTERNAL FB_StringHelper_Tests EXTENDS FB_TestSuite
VAR_INPUT
END_VAR
VAR_OUTPUT
END_VAR
VAR
END_VAR

Test01_StartsWith();
Test02_Join();
Test03_EndsWith();
Test05_Contains();
Test06_ToLowerCase_UnlimitedSize();
Test07_ToUpperCase_UnlimitedSize();

METHOD Test01_StartsWith
VAR_INPUT
END_VAR
TcUnit.TEST('Test01_StartsWith');

AssertFalse(StringHelper.StartsWith('I start with an "I"...','B'), 
	'The provided string does not start with B. Method should return FALSE.');
	
AssertTrue(StringHelper.StartsWith('I start with an "I"...','I'), 
	'The provided string start with I. Method should return TRUE..');

TcUnit.TEST_FINISHED();
END_METHOD

METHOD Test02_Join
VAR_INPUT
END_VAR

VAR
	sourceString	: Tc2_System.T_MaxString := 'My cats name is ';
END_VAR
TcUnit.TEST('Test02_Join');

StringHelper.Join(sourceString, 'Jerry');
AssertEquals_STRING('My cats name is Jerry', sourceString,
	'Joining 2 strings failed.');

TcUnit.TEST_FINISHED();
END_METHOD

METHOD Test03_EndsWith
VAR_INPUT
END_VAR

VAR
	testString	: STRING := 'I end with an A';
END_VAR
TcUnit.TEST('Test03_EndsWith');

AssertFalse(StringHelper.EndsWith(testString, 'B'),
	'Provided string does not end with "B"- returned value should be FALSE.');
AssertTrue(StringHelper.EndsWith(testString, 'A'),
	'Provided string ends with "A"- returned value should be TRUE.');
	
TcUnit.TEST_FINISHED();
END_METHOD

METHOD Test05_Contains
VAR_INPUT
END_VAR
VAR
	mainStringAsTmaxString		: Tc2_System.T_MaxString := 'asdfasdfadfasdfadfigsjcan you find mgndfkghdfghgdg!can you find me?';
	substringToFind_TmaxString	: STRING := 'can you find me';
	mainStringAsString300		: STRING(300) := 
		'abcdefghijklmnopqrstuvwxyzABCDEFGHIJKLMNOPQRSTUVWXYZ0123456789abcdefghijklmThis is the test sentence.nopqrstuvwxyzABCDEFGHIJKLMNOPQRSTUVWXYZ0123456789abcdefghijklmnopqrstuvwxyzABCDEFGHIJKLMNOPQRSTUVWXYZ0123456789abcdefghijklmnopqrstuvwxyz';
	substringToFind_String300	: STRING := 'This is the test sentence';	
	mainStringTmp				: STRING(300);
	position 					: DINT;
	test	: int;
END_VAR
TcUnit.TEST('Test05_Contains');

// T_MaxString tests

// doesen't contain
AssertFalse(StringHelper.FindStringWithin(mainStringAsTmaxString, 'test123', position => position),
	'String does not contain the provided substring.');
AssertEquals_DINT(0, position,
	'When string is not found, position should be 0');

// Upper case - fail
AssertFalse(StringHelper.FindStringWithin(mainStringAsTmaxString, StringHelper.ToUpperCase(substringToFind_TmaxString), position => position),
	'String should not be found, provided string is in upper case.');
AssertEquals_DINT(0, position,
	'When string is not found (upper case) , position should be 0');

// Contains	
AssertTrue(StringHelper.FindStringWithin(mainStringAsTmaxString, substringToFind_TmaxString, position => position),
	'String contains the provided substring, expected returned value should be TRUE.');
AssertEquals_DINT(52, position,
	'Incorrect position of the found substring.');
	

// Strings larger than T_MaxString tests
// Does not contain
AssertFalse(StringHelper.FindStringWithin(mainStringAsString300, 'test1234', position => position),
	'String300 - provided substring does not exist in the main string, expected FALSE.');
AssertEquals_DINT(0, position,
	'String300 - when substring is not found, expected position is 0.');
	
// Upper case - fail	
mainStringTmp := mainStringAsString300;
StringHelper.ToUpperCase_UnlimitedSize(mainStringTmp);
AssertFalse(StringHelper.FindStringWithin(mainStringAsTmaxString, mainStringTmp, position => position),
	'String300 upper case - String should not be found, provided string is in upper case.');
AssertEquals_DINT(0, position,
	'String300 upper case - When string is not found (upper case) , position should be 0');
	
// Lower case - fail
mainStringTmp := mainStringAsString300;
StringHelper.ToLowerCase_UnlimitedSize(mainStringTmp);
AssertFalse(StringHelper.FindStringWithin(mainStringAsTmaxString, mainStringTmp, position => position),
	'String300 lower case - String should not be found, provided string is in lower case.');
AssertEquals_DINT(0, position,
	'String300 lower case - When string is not found (lower case), position should be 0');
test := Tc2_Standard.FIND(mainStringAsString300, substringToFind_String300);
// Contains	
AssertTrue(StringHelper.FindStringWithin(mainStringAsString300, substringToFind_String300, position => position),
	'String contains the provided substring, expected returned value should be TRUE.');
AssertEquals_DINT(76, position,
	'Incorrect position of the found substring.');	
	
TcUnit.TEST_FINISHED();
END_METHOD

METHOD Test06_ToLowerCase_UnlimitedSize
VAR_INPUT
END_VAR
VAR_INST
	expectedResult	: STRING(300) := 'abcdefghijklmnopqrstuvwxyzabcdefghijklmnopqrstuvwxyz0123456789abcdefghijklmthis is the test sentence.nopqrstuvwxyzabcdefghijklmnopqrstuvwxyz0123456789abcdefghijklmnopqrstuvwxyzabcdefghijklmnopqrstuvwxyz0123456789abcdefghijklmnopqrstuvwxyz';
	providedString	: STRING(300) := 'ABCDEFGHIJKLMNOPQRSTUVWXYZABCDEFGHIJKLMNOPQRSTUVWXYZ0123456789ABCDEFGHIJKLMTHIS IS THE TEST SENTENCE.NOPQRSTUVWXYZABCDEFGHIJKLMNOPQRSTUVWXYZ0123456789ABCDEFGHIJKLMNOPQRSTUVWXYZABCDEFGHIJKLMNOPQRSTUVWXYZ0123456789ABCDEFGHIJKLMNOPQRSTUVWXYZ';
END_VAR
TcUnit.TEST('Test06_ToLowerCase_UnlimitedSize');

StringHelper.ToLowerCase_UnlimitedSize(providedString);
AssertEquals(expectedResult, providedString,
	'Incorrect conversion to lower case of string(300)');
	
TcUnit.TEST_FINISHED();
END_METHOD

METHOD Test07_ToUpperCase_UnlimitedSize
VAR_INPUT
END_VAR
VAR_INST
	providedString	: STRING(300) := 'abcdefghijklmnopqrstuvwxyzABCDEFGHIJKLMNOPQRSTUVWXYZ0123456789abcdefghijklmThis is the test sentence.nopqrstuvwxyzABCDEFGHIJKLMNOPQRSTUVWXYZ0123456789abcdefghijklmnopqrstuvwxyzABCDEFGHIJKLMNOPQRSTUVWXYZ0123456789abcdefghijklmnopqrstuvwxyz';
	expectedResult	: STRING(300) := 'ABCDEFGHIJKLMNOPQRSTUVWXYZABCDEFGHIJKLMNOPQRSTUVWXYZ0123456789ABCDEFGHIJKLMTHIS IS THE TEST SENTENCE.NOPQRSTUVWXYZABCDEFGHIJKLMNOPQRSTUVWXYZ0123456789ABCDEFGHIJKLMNOPQRSTUVWXYZABCDEFGHIJKLMNOPQRSTUVWXYZ0123456789ABCDEFGHIJKLMNOPQRSTUVWXYZ';
END_VAR
TcUnit.TEST('Test07_ToUpperCase_UnlimitedSize');

StringHelper.ToUpperCase_UnlimitedSize(providedString);
AssertEquals(expectedResult, providedString,
	'Incorrect conversion to upper case of string(300)');
	
TcUnit.TEST_FINISHED();
END_METHOD

END_FUNCTION_BLOCK
